                Waypoint Linea18_B: TCP in base x=-1149.609 y=625.735 z=110.055 mm, rx=1.1641 ry=-2.9058 rz=0.0105 rad; joints [-36.269, -18.655, 11.335, 7.818, -269.001, 0.894] deg; TCP offset x=0.411 y=-218.298 z=37.994 mm, rx=1.558 ry=-0.1255 rz=0.1212 rad
            Folder AB
              'desbaste_inicial'
              bajada_broca := p[0,0,-0.008,0,0,0]
              barrenos_menos1 := 19
              barreno_actual := 0
              Loop While (checkContinuously=false) expression=barreno_actual≤barrenos_menos1
                Folder Perforacion
                  MoveL speed 100 mm/s, acceleration 500 mm/s^2 (useActiveTCP=true) feature=Base
                    If barreno_actual≟6  or barreno_actual≟13
                      barreno_actual := barreno_actual+1
                    internos := interpolate_pose(Linea18_A, Linea18_B, barreno_actual/barrenos_menos1)
                    Waypoint Waypoint (Variable): variable=internos
                    'desbaste_inicial'
                    bajada_broca := p[0,0,-0.008,0,0,0]
                    bajada := p[0,0,0.008,0,0,0]
                    MoveDirectionNode (selectedDirection=ZMinus toolParams=0.1, 0.15)
                      Until DISTANCE (allowActions=false deceleration=3 distanceNodeType=STOP) Distance=0.071; motionParameters(blendRadius=0)
                    MoveDirectionNode (selectedDirection=ZMinus toolParams=0.001, 0.001)
                      Until TOOL_CONTACT_DETECTION (allowActions=false retraction=0 decelerationAcceleration=0.001 decelerationAngularAcceleration=34.906585)
                    Popup Message (haltProgram=false message=punto contacto alanzdo inputType=Text)
                    MoveDirectionNode (selectedDirection=ZPlus toolParams=0.003, 0.005)
                      Until DISTANCE (allowActions=false deceleration=3 distanceNodeType=STOP) Distance=0.002; motionParameters(blendRadius=0)
                    Wait Sleep waitTime=0.3
                    Set DigitalOutput pin=config_out[1]; digitalValue=1
                    Wait Sleep waitTime=0.3
                    SuppressedNode
                      Loop Counting (count=3) loopVariable=Loop_92
                        bajar := pose_add(get_actual_tcp_pose(), bajada_broca)
                        Waypoint Waypoint (Variable): motionParameters(jointSpeed=1.047198 jointAcceleration=1.396263 cartesianSpeed=0.001 cartesianAcceleration=0.005); variable=bajar
                        subir := pose_sub(get_actual_tcp_pose(), bajada_broca)
                        Waypoint Waypoint (Variable): motionParameters(jointSpeed=1.047198 jointAcceleration=1.396263 cartesianSpeed=0.005 cartesianAcceleration=0.01); variable=subir
                        bajada_broca := pose_sub(bajada_broca, bajada)
                    MoveDirectionNode (selectedDirection=ZPlus toolParams=0.1, 0.15)
                      Until DISTANCE (allowActions=false deceleration=3 distanceNodeType=STOP) Distance=0.08; motionParameters(blendRadius=0)
                    Set DigitalOutput pin=config_out[1]; digitalValue=0
                    barreno_actual := barreno_actual+1
                    SuppressedNode
                      Call Quitar_broca
                    SuppressedNode
                      Call Poner_broca
          Popup Message (haltProgram=false message=Linea18 con chica Terminada! inputType=Text)
      Folder Broca_1
        Folder Linea7
          Folder Marcar_puntos
            MoveL speed 100 mm/s, acceleration 500 mm/s^2 (useActiveTCP=true) feature=Base
              Waypoint Home2: TCP in base x=649.602 y=3.2 z=254.15 mm, rx=-2.4485 ry=-1.9662 rz=-0.0111 rad; joints [-199.372, -96.579, 116.673, -19.801, -286.041, 0.348] deg
              Waypoint Linea7_A: TCP in base x=737.913 y=-359.697 z=110.247 mm, rx=3.1319 ry=0.1866 rz=-0.0004 rad; joints [-210.915, -68.733, 100.688, -31.639, -226.901, 0.305] deg
              Folder bajada_comprobacion
                MoveDirectionNode (selectedDirection=ZMinus toolParams=0.1, 0.15)
                  Until DISTANCE (allowActions=false deceleration=3 distanceNodeType=STOP) Distance=0.071; motionParameters(blendRadius=0)
                MoveDirectionNode (selectedDirection=ZMinus toolParams=0.007, 0.007)
                  Until TOOL_CONTACT_DETECTION (allowActions=false retraction=0 decelerationAcceleration=0.02 decelerationAngularAcceleration=34.906585)
                MoveDirectionNode (selectedDirection=ZPlus toolParams=0.1, 0.15)
                  Until DISTANCE (allowActions=false deceleration=3 distanceNodeType=STOP) Distance=0.08; motionParameters(blendRadius=0)
              Waypoint Linea7_B: TCP in base x=783.713 y=-360.081 z=110.621 mm, rx=3.1319 ry=0.1866 rz=-0.0004 rad; joints [-209.138, -65.085, 95.206, -29.798, -225.12, 0.318] deg
              Folder bajada_comprobacion
                MoveDirectionNode (selectedDirection=ZMinus toolParams=0.1, 0.15)
                  Until DISTANCE (allowActions=false deceleration=3 distanceNodeType=STOP) Distance=0.071; motionParameters(blendRadius=0)
                MoveDirectionNode (selectedDirection=ZMinus toolParams=0.007, 0.007)
                  Until TOOL_CONTACT_DETECTION (allowActions=false retraction=0 decelerationAcceleration=0.02 decelerationAngularAcceleration=34.906585)
                MoveDirectionNode (selectedDirection=ZPlus toolParams=0.1, 0.15)
                  Until DISTANCE (allowActions=false deceleration=3 distanceNodeType=STOP) Distance=0.08; motionParameters(blendRadius=0)
          Folder AB
            'desbaste_inicial'
            bajada_broca := p[0,0,-0.008,0,0,0]
            barrenos_menos1 := 2
            barreno_actual := 1
            Loop While (checkContinuously=false) expression=barreno_actual≤barrenos_menos1
              Folder Perforacion
                MoveL speed 100 mm/s, acceleration 500 mm/s^2 (useActiveTCP=true) feature=Base
                  internos := interpolate_pose(Linea7_A, Linea7_B, barreno_actual/barrenos_menos1)
                  Waypoint Waypoint (Variable): variable=internos
                  'desbaste_inicial'
                  bajada_broca := p[0,0,-0.024,0,0,0]
                  bajada := p[0,0,0.024,0,0,0]
                  MoveDirectionNode (selectedDirection=ZMinus toolParams=0.1, 0.15)
                    Until DISTANCE (allowActions=false deceleration=3 distanceNodeType=STOP) Distance=0.071; motionParameters(blendRadius=0)
                  MoveDirectionNode (selectedDirection=ZMinus toolParams=0.007, 0.007)
                    Until TOOL_CONTACT_DETECTION (allowActions=false retraction=0 decelerationAcceleration=0.02 decelerationAngularAcceleration=34.906585)
                  Popup Message (haltProgram=false message=punto contacto alanzdo inputType=Text)
                  MoveDirectionNode (selectedDirection=ZPlus toolParams=0.015, 0.015)
                    Until DISTANCE (allowActions=false deceleration=3 distanceNodeType=STOP) Distance=0.007; motionParameters(blendRadius=0)
                  Wait Sleep waitTime=0.3
                  Set DigitalOutput pin=config_out[1]; digitalValue=1
                  Wait Sleep waitTime=0.3
                  Loop Counting (count=1) loopVariable(name=Loop_96)
                    bajar := pose_add(get_actual_tcp_pose(), bajada_broca)
                    Waypoint Waypoint (Variable): motionParameters(jointSpeed=1.047198 jointAcceleration=1.396263 cartesianSpeed=0.004 cartesianAcceleration=0.004); variable=bajar
                    subir := pose_sub(get_actual_tcp_pose(), bajada_broca)
                    MoveDirectionNode (selectedDirection=ZPlus toolParams=0.015, 0.015)
                      Until DISTANCE (allowActions=false deceleration=3 distanceNodeType=STOP) Distance=0.002; motionParameters(blendRadius=0)
                    Set DigitalOutput pin=config_out[1]; digitalValue=0
                    Waypoint Waypoint (Variable): motionParameters(jointSpeed=1.047198 jointAcceleration=1.396263 cartesianSpeed=0.015 cartesianAcceleration=0.015); variable=subir
                    bajada_broca := pose_sub(bajada_broca, bajada)
                  MoveDirectionNode (selectedDirection=ZPlus toolParams=0.1, 0.15)
                    Until DISTANCE (allowActions=false deceleration=3 distanceNodeType=STOP) Distance=0.08; motionParameters(blendRadius=0)
                  Set DigitalOutput pin=config_out[1]; digitalValue=0
                  barreno_actual := barreno_actual+1
                  Call Quitar_broca
                  Call Poner_broca
        Popup Message (haltProgram=false message=Linea7 con chica Terminada! inputType=Text)
        Folder Linea8
          Folder Marcar_puntos
            MoveL speed 100 mm/s, acceleration 500 mm/s^2 (useActiveTCP=true) feature=Base
              Waypoint Linea8_A: TCP in base x=886.283 y=-360.229 z=110.454 mm, rx=3.1315 ry=0.1865 rz=0.0006 rad; joints [-205.767, -56.675, 81.874, -24.901, -221.735, 0.344] deg
              Folder bajada_comprobacion
                MoveDirectionNode (selectedDirection=ZMinus toolParams=0.1, 0.15)
                  Until DISTANCE (allowActions=false deceleration=3 distanceNodeType=STOP) Distance=0.071; motionParameters(blendRadius=0)
                MoveDirectionNode (selectedDirection=ZMinus toolParams=0.007, 0.007)
                  Until TOOL_CONTACT_DETECTION (allowActions=false retraction=0 decelerationAcceleration=0.02 decelerationAngularAcceleration=34.906585)
                MoveDirectionNode (selectedDirection=ZPlus toolParams=0.1, 0.15)
                  Until DISTANCE (allowActions=false deceleration=3 distanceNodeType=STOP) Distance=0.08; motionParameters(blendRadius=0)
              Waypoint Linea8_B: TCP in base x=1009.987 y=-360.229 z=110.179 mm, rx=3.1315 ry=0.1865 rz=0.0006 rad; joints [-202.59, -45.403, 62.493, -16.778, -218.539, 0.367] deg
              Folder bajada_comprobacion
                MoveDirectionNode (selectedDirection=ZMinus toolParams=0.1, 0.15)
                  Until DISTANCE (allowActions=false deceleration=3 distanceNodeType=STOP) Distance=0.071; motionParameters(blendRadius=0)
                MoveDirectionNode (selectedDirection=ZMinus toolParams=0.007, 0.007)
                  Until TOOL_CONTACT_DETECTION (allowActions=false retraction=0 decelerationAcceleration=0.02 decelerationAngularAcceleration=34.906585)
                MoveDirectionNode (selectedDirection=ZPlus toolParams=0.1, 0.15)
                  Until DISTANCE (allowActions=false deceleration=3 distanceNodeType=STOP) Distance=0.08; motionParameters(blendRadius=0)
          Folder AB
            'desbaste_inicial'
            bajada_broca := p[0,0,-0.008,0,0,0]
            barrenos_menos1 := 5
            barreno_actual := 0
            Loop While (checkContinuously=false) expression=barreno_actual≤barrenos_menos1
              Folder Perforacion
                MoveL speed 100 mm/s, acceleration 500 mm/s^2 (useActiveTCP=true) feature=Base
                  internos := interpolate_pose(Linea8_A, Linea8_B, barreno_actual/barrenos_menos1)
                  Waypoint Waypoint (Variable): variable=internos
                  'desbaste_inicial'
                  bajada_broca := p[0,0,-0.024,0,0,0]
                  bajada := p[0,0,0.0024,0,0,0]
                  MoveDirectionNode (selectedDirection=ZMinus toolParams=0.1, 0.15)
                    Until DISTANCE (allowActions=false deceleration=3 distanceNodeType=STOP) Distance=0.071; motionParameters(blendRadius=0)
                  MoveDirectionNode (selectedDirection=ZMinus toolParams=0.007, 0.007)
                    Until TOOL_CONTACT_DETECTION (allowActions=false retraction=0 decelerationAcceleration=0.02 decelerationAngularAcceleration=34.906585)
                  Popup Message (haltProgram=false message=punto contacto alanzdo inputType=Text)
                  MoveDirectionNode (selectedDirection=ZPlus toolParams=0.015, 0.015)
                    Until DISTANCE (allowActions=false deceleration=3 distanceNodeType=STOP) Distance=0.007; motionParameters(blendRadius=0)
                  Wait Sleep waitTime=0.3
                  Set DigitalOutput pin=config_out[1]; digitalValue=1
                  Wait Sleep waitTime=0.3
                  Loop Counting (count=1) loopVariable(name=Loop_110)
                    bajar := pose_add(get_actual_tcp_pose(), bajada_broca)
                    Waypoint Waypoint (Variable): motionParameters(jointSpeed=1.047198 jointAcceleration=1.396263 cartesianSpeed=0.004 cartesianAcceleration=0.004); variable=bajar
                    subir := pose_sub(get_actual_tcp_pose(), bajada_broca)
                    MoveDirectionNode (selectedDirection=ZPlus toolParams=0.015, 0.015)
                      Until DISTANCE (allowActions=false deceleration=3 distanceNodeType=STOP) Distance=0.002; motionParameters(blendRadius=0)
                    Set DigitalOutput pin=config_out[1]; digitalValue=0
                    Waypoint Waypoint (Variable): motionParameters(jointSpeed=1.047198 jointAcceleration=1.396263 cartesianSpeed=0.015 cartesianAcceleration=0.015); variable=subir
                    bajada_broca := pose_sub(bajada_broca, bajada)
                  MoveDirectionNode (selectedDirection=ZPlus toolParams=0.1, 0.15)
                    Until DISTANCE (allowActions=false deceleration=3 distanceNodeType=STOP) Distance=0.08; motionParameters(blendRadius=0)
                  Set DigitalOutput pin=config_out[1]; digitalValue=0
                  barreno_actual := barreno_actual+1
                  Call Quitar_broca
                  Call Poner_broca
        Popup Message (haltProgram=false message=Linea8 con chica Terminada! inputType=Text)
        Folder Linea9
          Folder Marcar_puntos
            MoveL speed 100 mm/s, acceleration 500 mm/s^2 (useActiveTCP=true) feature=Base
              Waypoint Linea9_A: TCP in base x=1089.313 y=-360.631 z=110.237 mm, rx=3.1313 ry=0.1866 rz=0.0014 rad; joints [-200.952, -36.589, 46.349, -9.474, -216.885, 0.379] deg
              Folder bajada_comprobacion
                MoveDirectionNode (selectedDirection=ZMinus toolParams=0.1, 0.15)
                  Until DISTANCE (allowActions=false deceleration=3 distanceNodeType=STOP) Distance=0.071; motionParameters(blendRadius=0)
                MoveDirectionNode (selectedDirection=ZMinus toolParams=0.007, 0.007)
                  Until TOOL_CONTACT_DETECTION (allowActions=false retraction=0 decelerationAcceleration=0.02 decelerationAngularAcceleration=34.906585)
                MoveDirectionNode (selectedDirection=ZPlus toolParams=0.1, 0.15)
                  Until DISTANCE (allowActions=false deceleration=3 distanceNodeType=STOP) Distance=0.08; motionParameters(blendRadius=0)
              Waypoint Linea9_B: TCP in base x=1138.944 y=-360.869 z=110.826 mm, rx=3.1313 ry=0.1866 rz=0.0014 rad; joints [-200.044, -29.362, 32.524, -2.871, -215.958, 0.386] deg
              Folder bajada_comprobacion
                MoveDirectionNode (selectedDirection=ZMinus toolParams=0.1, 0.15)
                  Until DISTANCE (allowActions=false deceleration=3 distanceNodeType=STOP) Distance=0.071; motionParameters(blendRadius=0)
                MoveDirectionNode (selectedDirection=ZMinus toolParams=0.007, 0.007)
                  Until TOOL_CONTACT_DETECTION (allowActions=false retraction=0 decelerationAcceleration=0.02 decelerationAngularAcceleration=34.906585)
                MoveDirectionNode (selectedDirection=ZPlus toolParams=0.1, 0.15)
                  Until DISTANCE (allowActions=false deceleration=3 distanceNodeType=STOP) Distance=0.08; motionParameters(blendRadius=0)
          Folder AB
            'desbaste_inicial'
            bajada_broca := p[0,0,-0.008,0,0,0]
            barrenos_menos1 := 2
            barreno_actual := 0
            Loop While (checkContinuously=false) expression=barreno_actual≤barrenos_menos1
              Folder Perforacion
                MoveL speed 100 mm/s, acceleration 500 mm/s^2 (useActiveTCP=true) feature=Base
                  internos := interpolate_pose(Linea9_A, Linea9_B, barreno_actual/barrenos_menos1)
                  Waypoint Waypoint (Variable): variable=internos
                  'desbaste_inicial'
                  bajada_broca := p[0,0,-0.024,0,0,0]
                  bajada := p[0,0,0.024,0,0,0]
                  MoveDirectionNode (selectedDirection=ZMinus toolParams=0.1, 0.15)
                    Until DISTANCE (allowActions=false deceleration=3 distanceNodeType=STOP) Distance=0.071; motionParameters(blendRadius=0)
                  MoveDirectionNode (selectedDirection=ZMinus toolParams=0.007, 0.007)
                    Until TOOL_CONTACT_DETECTION (allowActions=false retraction=0 decelerationAcceleration=0.02 decelerationAngularAcceleration=34.906585)
                  Popup Message (haltProgram=false message=punto contacto alanzdo inputType=Text)
                  MoveDirectionNode (selectedDirection=ZPlus toolParams=0.015, 0.015)
                    Until DISTANCE (allowActions=false deceleration=3 distanceNodeType=STOP) Distance=0.007; motionParameters(blendRadius=0)
                  Wait Sleep waitTime=0.3
                  Set DigitalOutput pin=config_out[1]; digitalValue=1
                  Wait Sleep waitTime=0.3
                  Loop Counting (count=1) loopVariable(name=Loop_114)
                    bajar := pose_add(get_actual_tcp_pose(), bajada_broca)
                    Waypoint Waypoint (Variable): motionParameters(jointSpeed=1.047198 jointAcceleration=1.396263 cartesianSpeed=0.004 cartesianAcceleration=0.004); variable=bajar
                    subir := pose_sub(get_actual_tcp_pose(), bajada_broca)
                    MoveDirectionNode (selectedDirection=ZPlus toolParams=0.015, 0.015)
                      Until DISTANCE (allowActions=false deceleration=3 distanceNodeType=STOP) Distance=0.002; motionParameters(blendRadius=0)
                    Set DigitalOutput pin=config_out[1]; digitalValue=0
                    Waypoint Waypoint (Variable): motionParameters(jointSpeed=1.047198 jointAcceleration=1.396263 cartesianSpeed=0.015 cartesianAcceleration=0.015); variable=subir
                    bajada_broca := pose_sub(bajada_broca, bajada)
                  MoveDirectionNode (selectedDirection=ZPlus toolParams=0.1, 0.15)
                    Until DISTANCE (allowActions=false deceleration=3 distanceNodeType=STOP) Distance=0.08; motionParameters(blendRadius=0)
                  Set DigitalOutput pin=config_out[1]; digitalValue=0
                  barreno_actual := barreno_actual+1
                  Call Quitar_broca
                  Call Poner_broca
        Popup Message (haltProgram=false message=Linea9 con chica Terminada! inputType=Text)
        Folder Linea10
          Folder Marcar_puntos
            MoveL speed 100 mm/s, acceleration 500 mm/s^2 (useActiveTCP=true) feature=Base
              Waypoint Home2: TCP in base x=649.602 y=3.2 z=254.15 mm, rx=-2.4485 ry=-1.9662 rz=-0.0111 rad; joints [-199.372, -96.579, 116.673, -19.801, -286.041, 0.348] deg
              Waypoint Linea10_A: TCP in base x=620.978 y=-324.892 z=110.624 mm, rx=3.1274 ry=-0.2451 rz=-0.0041 rad; joints [-211.246, -75.766, 110.43, -34.284, -211.451, 0.322] deg; TCP offset x=0.411 y=-218.298 z=37.994 mm, rx=1.558 ry=-0.1255 rz=0.1212 rad
              Folder bajada_comprobacion
                MoveDirectionNode (selectedDirection=ZMinus toolParams=0.1, 0.15)
                  Until DISTANCE (allowActions=false deceleration=3 distanceNodeType=STOP) Distance=0.071; motionParameters(blendRadius=0)
                MoveDirectionNode (selectedDirection=ZMinus toolParams=0.007, 0.007)
                  Until TOOL_CONTACT_DETECTION (allowActions=false retraction=0 decelerationAcceleration=0.02 decelerationAngularAcceleration=34.906585)
                MoveDirectionNode (selectedDirection=ZPlus toolParams=0.1, 0.15)
                  Until DISTANCE (allowActions=false deceleration=3 distanceNodeType=STOP) Distance=0.08; motionParameters(blendRadius=0)
              Waypoint Linea10_B: TCP in base x=621.098 y=-276.98 z=110.32 mm, rx=3.1274 ry=-0.2451 rz=-0.0041 rad; joints [-207.342, -76.685, 111.673, -34.563, -207.548, 0.378] deg
              Folder bajada_comprobacion
                MoveDirectionNode (selectedDirection=ZMinus toolParams=0.1, 0.15)
                  Until DISTANCE (allowActions=false deceleration=3 distanceNodeType=STOP) Distance=0.071; motionParameters(blendRadius=0)
                MoveDirectionNode (selectedDirection=ZMinus toolParams=0.007, 0.007)
                  Until TOOL_CONTACT_DETECTION (allowActions=false retraction=0 decelerationAcceleration=0.02 decelerationAngularAcceleration=34.906585)
                MoveDirectionNode (selectedDirection=ZPlus toolParams=0.1, 0.15)
                  Until DISTANCE (allowActions=false deceleration=3 distanceNodeType=STOP) Distance=0.08; motionParameters(blendRadius=0)
          Folder AB
            'desbaste_inicial'
            bajada_broca := p[0,0,-0.008,0,0,0]
            barrenos_menos1 := 2
            barreno_actual := 0
            Loop While (checkContinuously=false) expression=barreno_actual≤barrenos_menos1
              Folder Perforacion
                MoveL speed 100 mm/s, acceleration 500 mm/s^2 (useActiveTCP=true) feature=Base
                  internos := interpolate_pose(Linea10_A, Linea10_B, barreno_actual/barrenos_menos1)
                  Waypoint Waypoint (Variable): variable=internos
                  'desbaste_inicial'
                  bajada_broca := p[0,0,-0.024,0,0,0]
                  bajada := p[0,0,0.024,0,0,0]
                  MoveDirectionNode (selectedDirection=ZMinus toolParams=0.1, 0.15)
                    Until DISTANCE (allowActions=false deceleration=3 distanceNodeType=STOP) Distance=0.071; motionParameters(blendRadius=0)
                  MoveDirectionNode (selectedDirection=ZMinus toolParams=0.007, 0.007)
                    Until TOOL_CONTACT_DETECTION (allowActions=false retraction=0 decelerationAcceleration=0.02 decelerationAngularAcceleration=34.906585)
                  Popup Message (haltProgram=false message=punto contacto alanzdo inputType=Text)
                  MoveDirectionNode (selectedDirection=ZPlus toolParams=0.015, 0.015)
                    Until DISTANCE (allowActions=false deceleration=3 distanceNodeType=STOP) Distance=0.007; motionParameters(blendRadius=0)
                  Wait Sleep waitTime=0.3
                  Set DigitalOutput pin=config_out[1]; digitalValue=1
                  Wait Sleep waitTime=0.3
                  Loop Counting (count=1) loopVariable(name=Loop_118)
                    bajar := pose_add(get_actual_tcp_pose(), bajada_broca)
                    Waypoint Waypoint (Variable): motionParameters(jointSpeed=1.047198 jointAcceleration=1.396263 cartesianSpeed=0.004 cartesianAcceleration=0.004); variable=bajar
                    subir := pose_sub(get_actual_tcp_pose(), bajada_broca)
                    MoveDirectionNode (selectedDirection=ZPlus toolParams=0.015, 0.015)
                      Until DISTANCE (allowActions=false deceleration=3 distanceNodeType=STOP) Distance=0.002; motionParameters(blendRadius=0)
                    Set DigitalOutput pin=config_out[1]; digitalValue=0
                    Waypoint Waypoint (Variable): motionParameters(jointSpeed=1.047198 jointAcceleration=1.396263 cartesianSpeed=0.015 cartesianAcceleration=0.015); variable=subir
                    bajada_broca := pose_sub(bajada_broca, bajada)
                  MoveDirectionNode (selectedDirection=ZPlus toolParams=0.1, 0.15)
                    Until DISTANCE (allowActions=false deceleration=3 distanceNodeType=STOP) Distance=0.08; motionParameters(blendRadius=0)
                  Set DigitalOutput pin=config_out[1]; digitalValue=0
                  barreno_actual := barreno_actual+1
                  SuppressedNode
                    Call Quitar_broca
                  SuppressedNode
                    Call Poner_broca
        Popup Message (haltProgram=false message=Linea10 con chica Terminada! inputType=Text)
        Folder Linea11
          Folder Marcar_puntos
            MoveL speed 100 mm/s, acceleration 500 mm/s^2 (useActiveTCP=true) feature=Base
              Waypoint Linea11_A: TCP in base x=623.455 y=-144.673 z=110.191 mm, rx=-2.632 ry=-1.7105 rz=-0.0086 rad; joints [-213.683, -89.957, 126.956, -36.551, -288.892, 0.32] deg
              Folder bajada_comprobacion
                MoveDirectionNode (selectedDirection=ZMinus toolParams=0.1, 0.15)
                  Until DISTANCE (allowActions=false deceleration=3 distanceNodeType=STOP) Distance=0.071; motionParameters(blendRadius=0)
                MoveDirectionNode (selectedDirection=ZMinus toolParams=0.007, 0.007)
                  Until TOOL_CONTACT_DETECTION (allowActions=false retraction=0 decelerationAcceleration=0.02 decelerationAngularAcceleration=34.906585)
                MoveDirectionNode (selectedDirection=ZPlus toolParams=0.1, 0.15)
                  Until DISTANCE (allowActions=false deceleration=3 distanceNodeType=STOP) Distance=0.08; motionParameters(blendRadius=0)
              Waypoint Linea11_B: TCP in base x=624.12 y=-90.095 z=110.354 mm, rx=-2.632 ry=-1.7105 rz=-0.0086 rad; joints [-207.683, -90.822, 127.793, -36.543, -282.892, 0.367] deg
              Folder bajada_comprobacion
                MoveDirectionNode (selectedDirection=ZMinus toolParams=0.1, 0.15)
                  Until DISTANCE (allowActions=false deceleration=3 distanceNodeType=STOP) Distance=0.071; motionParameters(blendRadius=0)
                MoveDirectionNode (selectedDirection=ZMinus toolParams=0.007, 0.007)
                  Until TOOL_CONTACT_DETECTION (allowActions=false retraction=0 decelerationAcceleration=0.02 decelerationAngularAcceleration=34.906585)
                MoveDirectionNode (selectedDirection=ZPlus toolParams=0.1, 0.15)
                  Until DISTANCE (allowActions=false deceleration=3 distanceNodeType=STOP) Distance=0.08; motionParameters(blendRadius=0)
          Folder AB
            'desbaste_inicial'
            bajada_broca := p[0,0,-0.008,0,0,0]
            barrenos_menos1 := 2
            barreno_actual := 0
            Loop While (checkContinuously=false) expression=barreno_actual≤barrenos_menos1
              Folder Perforacion
                MoveL speed 100 mm/s, acceleration 500 mm/s^2 (useActiveTCP=true) feature=Base
                  SuppressedNode
                    If barreno_actual≟5
                      barreno_actual := barreno_actual+1
                  internos := interpolate_pose(Linea11_A, Linea11_B, barreno_actual/barrenos_menos1)
                  Waypoint Waypoint (Variable): variable=internos
                  'desbaste_inicial'
                  bajada_broca := p[0,0,-0.024,0,0,0]
                  bajada := p[0,0,0.024,0,0,0]
                  MoveDirectionNode (selectedDirection=ZMinus toolParams=0.1, 0.15)
                    Until DISTANCE (allowActions=false deceleration=3 distanceNodeType=STOP) Distance=0.071; motionParameters(blendRadius=0)
                  MoveDirectionNode (selectedDirection=ZMinus toolParams=0.007, 0.007)
                    Until TOOL_CONTACT_DETECTION (allowActions=false retraction=0 decelerationAcceleration=0.02 decelerationAngularAcceleration=34.906585)
                  Popup Message (haltProgram=false message=punto contacto alanzdo inputType=Text)
                  MoveDirectionNode (selectedDirection=ZPlus toolParams=0.015, 0.015)
                    Until DISTANCE (allowActions=false deceleration=3 distanceNodeType=STOP) Distance=0.007; motionParameters(blendRadius=0)
                  Wait Sleep waitTime=0.3
                  Set DigitalOutput pin=config_out[1]; digitalValue=1
                  Wait Sleep waitTime=0.3
                  Loop Counting (count=1) loopVariable(name=Loop_122)
                    bajar := pose_add(get_actual_tcp_pose(), bajada_broca)
                    Waypoint Waypoint (Variable): motionParameters(jointSpeed=1.047198 jointAcceleration=1.396263 cartesianSpeed=0.004 cartesianAcceleration=0.004); variable=bajar
                    subir := pose_sub(get_actual_tcp_pose(), bajada_broca)
                    MoveDirectionNode (selectedDirection=ZPlus toolParams=0.015, 0.015)
                      Until DISTANCE (allowActions=false deceleration=3 distanceNodeType=STOP) Distance=0.002; motionParameters(blendRadius=0)
                    Set DigitalOutput pin=config_out[1]; digitalValue=0
                    Waypoint Waypoint (Variable): motionParameters(jointSpeed=1.047198 jointAcceleration=1.396263 cartesianSpeed=0.015 cartesianAcceleration=0.015); variable=subir
                    bajada_broca := pose_sub(bajada_broca, bajada)
                  MoveDirectionNode (selectedDirection=ZPlus toolParams=0.1, 0.15)
                    Until DISTANCE (allowActions=false deceleration=3 distanceNodeType=STOP) Distance=0.08; motionParameters(blendRadius=0)
                  Set DigitalOutput pin=config_out[1]; digitalValue=0
                  barreno_actual := barreno_actual+1
                  SuppressedNode
                    Call Quitar_broca
                  SuppressedNode
                    Call Poner_broca
        Popup Message (haltProgram=false message=Linea11 con chica Terminada! inputType=Text)
        Folder Linea12
          Folder Marcar_puntos
            MoveL speed 100 mm/s, acceleration 500 mm/s^2 (useActiveTCP=true) feature=Base
              Waypoint Linea12_A: TCP in base x=624.141 y=-66.274 z=110.335 mm, rx=-2.6321 ry=-1.7106 rz=-0.0087 rad; joints [-204.939, -91.033, 128.004, -36.559, -280.152, 0.387] deg
              Folder bajada_comprobacion
                MoveDirectionNode (selectedDirection=ZMinus toolParams=0.1, 0.15)
                  Until DISTANCE (allowActions=false deceleration=3 distanceNodeType=STOP) Distance=0.071; motionParameters(blendRadius=0)
                MoveDirectionNode (selectedDirection=ZMinus toolParams=0.007, 0.007)
                  Until TOOL_CONTACT_DETECTION (allowActions=false retraction=0 decelerationAcceleration=0.02 decelerationAngularAcceleration=34.906585)
                MoveDirectionNode (selectedDirection=ZPlus toolParams=0.1, 0.15)
                  Until DISTANCE (allowActions=false deceleration=3 distanceNodeType=STOP) Distance=0.08; motionParameters(blendRadius=0)
              Waypoint Linea12_B: TCP in base x=625.005 y=106.664 z=110.181 mm, rx=-2.6321 ry=-1.7106 rz=-0.0087 rad; joints [-183.741, -88.918, 125.907, -36.601, -258.955, 0.536] deg
              Folder bajada_comprobacion
                MoveDirectionNode (selectedDirection=ZMinus toolParams=0.1, 0.15)
                  Until DISTANCE (allowActions=false deceleration=3 distanceNodeType=STOP) Distance=0.071; motionParameters(blendRadius=0)
                MoveDirectionNode (selectedDirection=ZMinus toolParams=0.007, 0.007)
                  Until TOOL_CONTACT_DETECTION (allowActions=false retraction=0 decelerationAcceleration=0.02 decelerationAngularAcceleration=34.906585)
                MoveDirectionNode (selectedDirection=ZPlus toolParams=0.1, 0.15)
                  Until DISTANCE (allowActions=false deceleration=3 distanceNodeType=STOP) Distance=0.08; motionParameters(blendRadius=0)
          Folder AB
            'desbaste_inicial'
            bajada_broca := p[0,0,-0.008,0,0,0]
            barrenos_menos1 := 7
            barreno_actual := 0
            Loop While (checkContinuously=false) expression=barreno_actual≤barrenos_menos1
              Folder Perforacion
                MoveL speed 100 mm/s, acceleration 500 mm/s^2 (useActiveTCP=true) feature=Base
                  If barreno_actual≟2
                    barreno_actual := barreno_actual+1
                  internos := interpolate_pose(Linea12_A, Linea12_B, barreno_actual/barrenos_menos1)
                  Waypoint Waypoint (Variable): variable=internos
                  'desbaste_inicial'
                  bajada_broca := p[0,0,-0.024,0,0,0]
                  bajada := p[0,0,0.024,0,0,0]
                  MoveDirectionNode (selectedDirection=ZMinus toolParams=0.1, 0.15)
                    Until DISTANCE (allowActions=false deceleration=3 distanceNodeType=STOP) Distance=0.071; motionParameters(blendRadius=0)
                  MoveDirectionNode (selectedDirection=ZMinus toolParams=0.007, 0.007)
                    Until TOOL_CONTACT_DETECTION (allowActions=false retraction=0 decelerationAcceleration=0.02 decelerationAngularAcceleration=34.906585)
                  Popup Message (haltProgram=false message=punto contacto alanzdo inputType=Text)
                  MoveDirectionNode (selectedDirection=ZPlus toolParams=0.015, 0.015)
                    Until DISTANCE (allowActions=false deceleration=3 distanceNodeType=STOP) Distance=0.002; motionParameters(blendRadius=0)
                  Wait Sleep waitTime=0.3
                  Set DigitalOutput pin=config_out[1]; digitalValue=1
                  Wait Sleep waitTime=0.3
                  Loop Counting (count=1) loopVariable(name=Loop_126)
                    bajar := pose_add(get_actual_tcp_pose(), bajada_broca)
                    Waypoint Waypoint (Variable): motionParameters(jointSpeed=1.047198 jointAcceleration=1.396263 cartesianSpeed=0.004 cartesianAcceleration=0.004); variable=bajar
                    subir := pose_sub(get_actual_tcp_pose(), bajada_broca)
                    MoveDirectionNode (selectedDirection=ZPlus toolParams=0.015, 0.015)
                      Until DISTANCE (allowActions=false deceleration=3 distanceNodeType=STOP) Distance=0.002; motionParameters(blendRadius=0)
                    Set DigitalOutput pin=config_out[1]; digitalValue=0
                    Waypoint Waypoint (Variable): motionParameters(jointSpeed=1.047198 jointAcceleration=1.396263 cartesianSpeed=0.015 cartesianAcceleration=0.015); variable=subir
                    bajada_broca := pose_sub(bajada_broca, bajada)
                  MoveDirectionNode (selectedDirection=ZPlus toolParams=0.1, 0.15)
                    Until DISTANCE (allowActions=false deceleration=3 distanceNodeType=STOP) Distance=0.08; motionParameters(blendRadius=0)
                  Set DigitalOutput pin=config_out[1]; digitalValue=0
                  barreno_actual := barreno_actual+1
                  SuppressedNode
                    Call Quitar_broca
                  SuppressedNode
                    Call Poner_broca
        Popup Message (haltProgram=false message=Linea12 con chica Terminada! inputType=Text)
        Folder Linea13
          Folder Marcar_puntos
            MoveL speed 100 mm/s, acceleration 500 mm/s^2 (useActiveTCP=true) feature=Base
              Waypoint Linea13_A: TCP in base x=625.493 y=262.479 z=110.355 mm, rx=-2.6325 ry=-1.7109 rz=-0.0101 rad; joints [-165.949, -82.781, 119.173, -36.043, -241.164, 0.656] deg
              Folder bajada_comprobacion
                MoveDirectionNode (selectedDirection=ZMinus toolParams=0.1, 0.15)
                  Until DISTANCE (allowActions=false deceleration=3 distanceNodeType=STOP) Distance=0.071; motionParameters(blendRadius=0)
                MoveDirectionNode (selectedDirection=ZMinus toolParams=0.007, 0.007)
                  Until TOOL_CONTACT_DETECTION (allowActions=false retraction=0 decelerationAcceleration=0.02 decelerationAngularAcceleration=34.906585)
                MoveDirectionNode (selectedDirection=ZPlus toolParams=0.1, 0.15)
                  Until DISTANCE (allowActions=false deceleration=3 distanceNodeType=STOP) Distance=0.08; motionParameters(blendRadius=0)
              Waypoint Linea13_B: TCP in base x=625.493 y=318.857 z=110.132 mm, rx=-2.6325 ry=-1.7109 rz=-0.0101 rad; joints [-160.355, -79.919, 115.767, -35.483, -235.569, 0.699] deg
              Folder bajada_comprobacion
                MoveDirectionNode (selectedDirection=ZMinus toolParams=0.1, 0.15)
                  Until DISTANCE (allowActions=false deceleration=3 distanceNodeType=STOP) Distance=0.071; motionParameters(blendRadius=0)
                MoveDirectionNode (selectedDirection=ZMinus toolParams=0.007, 0.007)
                  Until TOOL_CONTACT_DETECTION (allowActions=false retraction=0 decelerationAcceleration=0.02 decelerationAngularAcceleration=34.906585)
                MoveDirectionNode (selectedDirection=ZPlus toolParams=0.1, 0.15)
                  Until DISTANCE (allowActions=false deceleration=3 distanceNodeType=STOP) Distance=0.08; motionParameters(blendRadius=0)
          Folder AB
            'desbaste_inicial'
            bajada_broca := p[0,0,-0.008,0,0,0]
            barrenos_menos1 := 2
            barreno_actual := 0
            Loop While (checkContinuously=false) expression=barreno_actual≤barrenos_menos1
              Folder Perforacion
                MoveL speed 100 mm/s, acceleration 500 mm/s^2 (useActiveTCP=true) feature=Base
                  SuppressedNode
                    If barreno_actual≟2
                      barreno_actual := barreno_actual+1
                  internos := interpolate_pose(Linea13_A, Linea13_B, barreno_actual/barrenos_menos1)
                  Waypoint Waypoint (Variable): variable=internos
                  'desbaste_inicial'
                  bajada_broca := p[0,0,-0.024,0,0,0]
                  bajada := p[0,0,0.024,0,0,0]
                  MoveDirectionNode (selectedDirection=ZMinus toolParams=0.1, 0.15)
                    Until DISTANCE (allowActions=false deceleration=3 distanceNodeType=STOP) Distance=0.071; motionParameters(blendRadius=0)
                  MoveDirectionNode (selectedDirection=ZMinus toolParams=0.007, 0.007)
                    Until TOOL_CONTACT_DETECTION (allowActions=false retraction=0 decelerationAcceleration=0.02 decelerationAngularAcceleration=34.906585)
                  Popup Message (haltProgram=false message=punto contacto alanzdo inputType=Text)
                  MoveDirectionNode (selectedDirection=ZPlus toolParams=0.015, 0.015)
                    Until DISTANCE (allowActions=false deceleration=3 distanceNodeType=STOP) Distance=0.002; motionParameters(blendRadius=0)
                  Wait Sleep waitTime=0.3
                  Set DigitalOutput pin=config_out[1]; digitalValue=1
                  Wait Sleep waitTime=0.3
                  Loop Counting (count=1) loopVariable(name=Loop_129)
                    bajar := pose_add(get_actual_tcp_pose(), bajada_broca)
                    Waypoint Waypoint (Variable): motionParameters(jointSpeed=1.047198 jointAcceleration=1.396263 cartesianSpeed=0.004 cartesianAcceleration=0.004); variable=bajar
                    subir := pose_sub(get_actual_tcp_pose(), bajada_broca)
                    MoveDirectionNode (selectedDirection=ZPlus toolParams=0.015, 0.015)
                      Until DISTANCE (allowActions=false deceleration=3 distanceNodeType=STOP) Distance=0.002; motionParameters(blendRadius=0)
                    Set DigitalOutput pin=config_out[1]; digitalValue=0
                    Waypoint Waypoint (Variable): motionParameters(jointSpeed=1.047198 jointAcceleration=1.396263 cartesianSpeed=0.015 cartesianAcceleration=0.015); variable=subir
                    bajada_broca := pose_sub(bajada_broca, bajada)
                  MoveDirectionNode (selectedDirection=ZPlus toolParams=0.1, 0.15)
                    Until DISTANCE (allowActions=false deceleration=3 distanceNodeType=STOP) Distance=0.08; motionParameters(blendRadius=0)
                  Set DigitalOutput pin=config_out[1]; digitalValue=0
                  barreno_actual := barreno_actual+1
                  SuppressedNode
                    Call Quitar_broca
                  SuppressedNode
                    Call Poner_broca
        Popup Message (haltProgram=false message=Linea13 con chica Terminada! inputType=Text)
        Folder Linea14
          Folder Marcar_puntos
            MoveL speed 100 mm/s, acceleration 500 mm/s^2 (useActiveTCP=true) feature=Base
              Waypoint Linea14_A: TCP in base x=625.749 y=343.505 z=110.091 mm, rx=-2.6326 ry=-1.7111 rz=-0.011 rad; joints [-158.078, -78.594, 114.13, -35.197, -233.295, 0.717] deg
              barrenos_hechos := 0
              Folder bajada_comprobacion
                MoveDirectionNode (selectedDirection=ZMinus toolParams=0.1, 0.15)
                  Until DISTANCE (allowActions=false deceleration=3 distanceNodeType=STOP) Distance=0.071; motionParameters(blendRadius=0)
                MoveDirectionNode (selectedDirection=ZMinus toolParams=0.007, 0.007)
                  Until TOOL_CONTACT_DETECTION (allowActions=false retraction=0 decelerationAcceleration=0.02 decelerationAngularAcceleration=34.906585)
                MoveDirectionNode (selectedDirection=ZPlus toolParams=0.1, 0.15)
                  Until DISTANCE (allowActions=false deceleration=3 distanceNodeType=STOP) Distance=0.08; motionParameters(blendRadius=0)
              Waypoint Linea14_B: TCP in base x=626.023 y=485.153 z=110.594 mm, rx=-2.6326 ry=-1.7111 rz=-0.011 rad; joints [-146.753, -70.37, 102.998, -32.234, -221.967, 0.818] deg
              Folder bajada_comprobacion
                MoveDirectionNode (selectedDirection=ZMinus toolParams=0.1, 0.15)
                  Until DISTANCE (allowActions=false deceleration=3 distanceNodeType=STOP) Distance=0.071; motionParameters(blendRadius=0)
                MoveDirectionNode (selectedDirection=ZMinus toolParams=0.007, 0.007)
                  Until TOOL_CONTACT_DETECTION (allowActions=false retraction=0 decelerationAcceleration=0.02 decelerationAngularAcceleration=34.906585)
                MoveDirectionNode (selectedDirection=ZPlus toolParams=0.1, 0.15)
                  Until DISTANCE (allowActions=false deceleration=3 distanceNodeType=STOP) Distance=0.08; motionParameters(blendRadius=0)
          Folder AB
            'desbaste_inicial'
            bajada_broca := p[0,0,-0.008,0,0,0]
            barrenos_menos1 := 5
            barreno_actual := 0
            Loop While (checkContinuously=false) expression=barreno_actual≤barrenos_menos1
              Folder Perforacion
                MoveL speed 100 mm/s, acceleration 500 mm/s^2 (useActiveTCP=true) feature=Base
                  If barreno_actual≟3
                    barreno_actual := barreno_actual+1
                  internos := interpolate_pose(Linea14_A, Linea14_B, barreno_actual/barrenos_menos1)
                  Waypoint Waypoint (Variable): variable=internos
                  'desbaste_inicial'
                  bajada_broca := p[0,0,-0.024,0,0,0]
                  bajada := p[0,0,0.024,0,0,0]
                  MoveDirectionNode (selectedDirection=ZMinus toolParams=0.1, 0.15)
                    Until DISTANCE (allowActions=false deceleration=3 distanceNodeType=STOP) Distance=0.071; motionParameters(blendRadius=0)
                  MoveDirectionNode (selectedDirection=ZMinus toolParams=0.007, 0.007)
                    Until TOOL_CONTACT_DETECTION (allowActions=false retraction=0 decelerationAcceleration=0.02 decelerationAngularAcceleration=34.906585)
                  Popup Message (haltProgram=false message=punto contacto alanzdo inputType=Text)
                  MoveDirectionNode (selectedDirection=ZPlus toolParams=0.015, 0.015)
                    Until DISTANCE (allowActions=false deceleration=3 distanceNodeType=STOP) Distance=0.002; motionParameters(blendRadius=0)
                  Wait Sleep waitTime=0.3
                  Set DigitalOutput pin=config_out[1]; digitalValue=1
                  Wait Sleep waitTime=0.3
                  Loop Counting (count=1) loopVariable(name=Loop_131)
                    bajar := pose_add(get_actual_tcp_pose(), bajada_broca)
                    Waypoint Waypoint (Variable): motionParameters(jointSpeed=1.047198 jointAcceleration=1.396263 cartesianSpeed=0.004 cartesianAcceleration=0.004); variable=bajar
                    subir := pose_sub(get_actual_tcp_pose(), bajada_broca)
                    MoveDirectionNode (selectedDirection=ZPlus toolParams=0.015, 0.015)
                      Until DISTANCE (allowActions=false deceleration=3 distanceNodeType=STOP) Distance=0.002; motionParameters(blendRadius=0)
                    Set DigitalOutput pin=config_out[1]; digitalValue=0
                    Waypoint Waypoint (Variable): motionParameters(jointSpeed=1.047198 jointAcceleration=1.396263 cartesianSpeed=0.015 cartesianAcceleration=0.015); variable=subir
                    bajada_broca := pose_sub(bajada_broca, bajada)
                  MoveDirectionNode (selectedDirection=ZPlus toolParams=0.1, 0.15)
                    Until DISTANCE (allowActions=false deceleration=3 distanceNodeType=STOP) Distance=0.08; motionParameters(blendRadius=0)
                  Set DigitalOutput pin=config_out[1]; digitalValue=0
                  barreno_actual := barreno_actual+1
                  SuppressedNode
                    Call Quitar_broca
                  SuppressedNode
                    Call Poner_broca
        Popup Message (haltProgram=false message=Linea14 con chica Terminada! inputType=Text)
        Folder Linea15
          Folder Marcar_puntos
            MoveL speed 100 mm/s, acceleration 500 mm/s^2 (useActiveTCP=true) feature=Base
              Waypoint Linea15_A: TCP in base x=626.307 y=508.675 z=110.445 mm, rx=-2.6326 ry=-1.7111 rz=-0.011 rad; joints [-145.159, -68.884, 100.875, -31.585, -220.372, 0.835] deg
              barrenos_hechos := 0
              Folder bajada_comprobacion
                MoveDirectionNode (selectedDirection=ZMinus toolParams=0.1, 0.15)
                  Until DISTANCE (allowActions=false deceleration=3 distanceNodeType=STOP) Distance=0.071; motionParameters(blendRadius=0)
                MoveDirectionNode (selectedDirection=ZMinus toolParams=0.007, 0.007)
                  Until TOOL_CONTACT_DETECTION (allowActions=false retraction=0 decelerationAcceleration=0.02 decelerationAngularAcceleration=34.906585)
                MoveDirectionNode (selectedDirection=ZPlus toolParams=0.1, 0.15)
                  Until DISTANCE (allowActions=false deceleration=3 distanceNodeType=STOP) Distance=0.08; motionParameters(blendRadius=0)
              Waypoint Linea15_B: TCP in base x=626.328 y=587.416 z=110.05 mm, rx=-2.6327 ry=-1.711 rz=-0.011 rad; joints [-140.277, -63.781, 93.264, -29.039, -215.483, 0.889] deg
              Folder bajada_comprobacion
                MoveDirectionNode (selectedDirection=ZMinus toolParams=0.1, 0.15)
                  Until DISTANCE (allowActions=false deceleration=3 distanceNodeType=STOP) Distance=0.071; motionParameters(blendRadius=0)
                MoveDirectionNode (selectedDirection=ZMinus toolParams=0.007, 0.007)
                  Until TOOL_CONTACT_DETECTION (allowActions=false retraction=0 decelerationAcceleration=0.02 decelerationAngularAcceleration=34.906585)
                MoveDirectionNode (selectedDirection=ZPlus toolParams=0.1, 0.15)
                  Until DISTANCE (allowActions=false deceleration=3 distanceNodeType=STOP) Distance=0.08; motionParameters(blendRadius=0)
          Folder AB
            'desbaste_inicial'
            bajada_broca := p[0,0,-0.008,0,0,0]
            barrenos_menos1 := 3
            barreno_actual := 0
            Loop While (checkContinuously=false) expression=barreno_actual≤barrenos_menos1
              Folder Perforacion
                MoveL speed 100 mm/s, acceleration 500 mm/s^2 (useActiveTCP=true) feature=Base
                  SuppressedNode
                    If barreno_actual≟3
                      barreno_actual := barreno_actual+1
                  internos := interpolate_pose(Linea15_A, Linea15_B, barreno_actual/barrenos_menos1)
                  Waypoint Waypoint (Variable): variable=internos
                  'desbaste_inicial'
                  bajada_broca := p[0,0,-0.024,0,0,0]
                  bajada := p[0,0,0.024,0,0,0]
                  MoveDirectionNode (selectedDirection=ZMinus toolParams=0.1, 0.15)
                    Until DISTANCE (allowActions=false deceleration=3 distanceNodeType=STOP) Distance=0.071; motionParameters(blendRadius=0)
                  MoveDirectionNode (selectedDirection=ZMinus toolParams=0.007, 0.007)
                    Until TOOL_CONTACT_DETECTION (allowActions=false retraction=0 decelerationAcceleration=0.02 decelerationAngularAcceleration=34.906585)
                  Popup Message (haltProgram=false message=punto contacto alanzdo inputType=Text)
                  MoveDirectionNode (selectedDirection=ZPlus toolParams=0.015, 0.015)
                    Until DISTANCE (allowActions=false deceleration=3 distanceNodeType=STOP) Distance=0.002; motionParameters(blendRadius=0)
                  Wait Sleep waitTime=0.3
                  Set DigitalOutput pin=config_out[1]; digitalValue=1
                  Wait Sleep waitTime=0.3
                  Loop Counting (count=1) loopVariable(name=Loop_133)
                    bajar := pose_add(get_actual_tcp_pose(), bajada_broca)
                    Waypoint Waypoint (Variable): motionParameters(jointSpeed=1.047198 jointAcceleration=1.396263 cartesianSpeed=0.004 cartesianAcceleration=0.004); variable=bajar
                    subir := pose_sub(get_actual_tcp_pose(), bajada_broca)
                    MoveDirectionNode (selectedDirection=ZPlus toolParams=0.015, 0.015)
                      Until DISTANCE (allowActions=false deceleration=3 distanceNodeType=STOP) Distance=0.002; motionParameters(blendRadius=0)
                    Set DigitalOutput pin=config_out[1]; digitalValue=0
                    Waypoint Waypoint (Variable): motionParameters(jointSpeed=1.047198 jointAcceleration=1.396263 cartesianSpeed=0.015 cartesianAcceleration=0.015); variable=subir
                    bajada_broca := pose_sub(bajada_broca, bajada)
                  MoveDirectionNode (selectedDirection=ZPlus toolParams=0.1, 0.15)
                    Until DISTANCE (allowActions=false deceleration=3 distanceNodeType=STOP) Distance=0.08; motionParameters(blendRadius=0)
                  Set DigitalOutput pin=config_out[1]; digitalValue=0
                  barreno_actual := barreno_actual+1
                  SuppressedNode
                    Call Quitar_broca
                  SuppressedNode
                    Call Poner_broca
        Popup Message (haltProgram=false message=Linea15 con chica Terminada! inputType=Text)
        Folder Linea16
          Folder Marcar_puntos
            MoveL speed 100 mm/s, acceleration 500 mm/s^2 (useActiveTCP=true) feature=Base
              Waypoint Linea16_A referenceName=Linea16_A: TCP in base x=464.714 y=611.413 z=110.697 mm, rx=-1.5443 ry=-2.7321 rz=-0.0069 rad; joints [-140.663, -77.848, 113.101, -34.922, -270.882, 0.394] deg; TCP offset x=0.411 y=-218.298 z=37.994 mm, rx=1.558 ry=-0.1255 rz=0.1212 rad
              Folder bajada_comprobacion
                MoveDirectionNode (selectedDirection=ZMinus toolParams=0.1, 0.15)
                  Until DISTANCE (allowActions=false deceleration=3 distanceNodeType=STOP) Distance=0.071; motionParameters(blendRadius=0)
                MoveDirectionNode (selectedDirection=ZMinus toolParams=0.007, 0.007)
                  Until TOOL_CONTACT_DETECTION (allowActions=false retraction=0 decelerationAcceleration=0.02 decelerationAngularAcceleration=34.906585)
                MoveDirectionNode (selectedDirection=ZPlus toolParams=0.1, 0.15)
                  Until DISTANCE (allowActions=false deceleration=3 distanceNodeType=STOP) Distance=0.08; motionParameters(blendRadius=0)
              Waypoint Linea16_B: TCP in base x=487.741 y=611.018 z=110.415 mm, rx=-1.5443 ry=-2.7321 rz=-0.0069 rad; joints [-142.061, -76.715, 111.675, -34.628, -272.279, 0.386] deg
              Folder bajada_comprobacion
                MoveDirectionNode (selectedDirection=ZMinus toolParams=0.1, 0.15)
                  Until DISTANCE (allowActions=false deceleration=3 distanceNodeType=STOP) Distance=0.071; motionParameters(blendRadius=0)
                MoveDirectionNode (selectedDirection=ZMinus toolParams=0.007, 0.007)
                  Until TOOL_CONTACT_DETECTION (allowActions=false retraction=0 decelerationAcceleration=0.02 decelerationAngularAcceleration=34.906585)
                MoveDirectionNode (selectedDirection=ZPlus toolParams=0.1, 0.15)
                  Until DISTANCE (allowActions=false deceleration=3 distanceNodeType=STOP) Distance=0.08; motionParameters(blendRadius=0)
          Folder AB
            'desbaste_inicial'
            bajada_broca := p[0,0,-0.008,0,0,0]
            barrenos_menos1 := 1
            barreno_actual := 0
            Loop While (checkContinuously=false) expression=barreno_actual≤barrenos_menos1
              Folder Perforacion
                MoveL speed 100 mm/s, acceleration 500 mm/s^2 (useActiveTCP=true) feature=Base
                  SuppressedNode
                    If barreno_actual≟3
                      barreno_actual := barreno_actual+1
                  internos := interpolate_pose(Linea16_A, Linea16_B, barreno_actual/barrenos_menos1)
                  Waypoint Waypoint (Variable): variable=internos
                  'desbaste_inicial'
                  bajada_broca := p[0,0,-0.024,0,0,0]
                  bajada := p[0,0,0.024,0,0,0]
                  MoveDirectionNode (selectedDirection=ZMinus toolParams=0.1, 0.15)
                    Until DISTANCE (allowActions=false deceleration=3 distanceNodeType=STOP) Distance=0.071; motionParameters(blendRadius=0)
                  MoveDirectionNode (selectedDirection=ZMinus toolParams=0.007, 0.007)
                    Until TOOL_CONTACT_DETECTION (allowActions=false retraction=0 decelerationAcceleration=0.02 decelerationAngularAcceleration=34.906585)
                  Popup Message (haltProgram=false message=punto contacto alanzdo inputType=Text)
                  MoveDirectionNode (selectedDirection=ZPlus toolParams=0.015, 0.015)
                    Until DISTANCE (allowActions=false deceleration=3 distanceNodeType=STOP) Distance=0.007; motionParameters(blendRadius=0)
                  Wait Sleep waitTime=0.3
                  Set DigitalOutput pin=config_out[1]; digitalValue=1
                  Wait Sleep waitTime=0.3
                  Loop Counting (count=1) loopVariable(name=Loop_135)
                    bajar := pose_add(get_actual_tcp_pose(), bajada_broca)
                    Waypoint Waypoint (Variable): motionParameters(jointSpeed=1.047198 jointAcceleration=1.396263 cartesianSpeed=0.004 cartesianAcceleration=0.004); variable=bajar
                    subir := pose_sub(get_actual_tcp_pose(), bajada_broca)
                    MoveDirectionNode (selectedDirection=ZPlus toolParams=0.015, 0.015)
                      Until DISTANCE (allowActions=false deceleration=3 distanceNodeType=STOP) Distance=0.002; motionParameters(blendRadius=0)
                    Set DigitalOutput pin=config_out[1]; digitalValue=0
                    Waypoint Waypoint (Variable): motionParameters(jointSpeed=1.047198 jointAcceleration=1.396263 cartesianSpeed=0.015 cartesianAcceleration=0.015); variable=subir
                    bajada_broca := pose_sub(bajada_broca, bajada)
                  MoveDirectionNode (selectedDirection=ZPlus toolParams=0.1, 0.15)
                    Until DISTANCE (allowActions=false deceleration=3 distanceNodeType=STOP) Distance=0.08; motionParameters(blendRadius=0)
                  Set DigitalOutput pin=config_out[1]; digitalValue=0
                  barreno_actual := barreno_actual+1
                  SuppressedNode
                    Call Quitar_broca
                  SuppressedNode
                    Call Poner_broca
        Popup Message (haltProgram=false message=Linea16 con chica Terminada! inputType=Text)
        Folder Linea17
          Folder Marcar_puntos
            MoveL speed 100 mm/s, acceleration 500 mm/s^2 (useActiveTCP=true) feature=Base
              Waypoint Linea17_A: TCP in base x=517.384 y=611.103 z=110.729 mm, rx=-1.5448 ry=-2.7327 rz=-0.0099 rad; joints [-143.713, -75.238, 109.731, -34.279, -273.925, 0.383] deg
              Folder bajada_comprobacion
                MoveDirectionNode (selectedDirection=ZMinus toolParams=0.1, 0.15)
                  Until DISTANCE (allowActions=false deceleration=3 distanceNodeType=STOP) Distance=0.071; motionParameters(blendRadius=0)
                MoveDirectionNode (selectedDirection=ZMinus toolParams=0.007, 0.007)
                  Until TOOL_CONTACT_DETECTION (allowActions=false retraction=0 decelerationAcceleration=0.02 decelerationAngularAcceleration=34.906585)
                MoveDirectionNode (selectedDirection=ZPlus toolParams=0.1, 0.15)
                  Until DISTANCE (allowActions=false deceleration=3 distanceNodeType=STOP) Distance=0.08; motionParameters(blendRadius=0)
              Waypoint Linea17_B: TCP in base x=569.253 y=610.697 z=110.46 mm, rx=-1.5448 ry=-2.7327 rz=-0.0099 rad; joints [-146.385, -72.438, 105.956, -33.3, -276.596, 0.373] deg
              Folder bajada_comprobacion
                MoveDirectionNode (selectedDirection=ZMinus toolParams=0.1, 0.15)
                  Until DISTANCE (allowActions=false deceleration=3 distanceNodeType=STOP) Distance=0.071; motionParameters(blendRadius=0)
                MoveDirectionNode (selectedDirection=ZMinus toolParams=0.007, 0.007)
                  Until TOOL_CONTACT_DETECTION (allowActions=false retraction=0 decelerationAcceleration=0.02 decelerationAngularAcceleration=34.906585)
                MoveDirectionNode (selectedDirection=ZPlus toolParams=0.1, 0.15)
                  Until DISTANCE (allowActions=false deceleration=3 distanceNodeType=STOP) Distance=0.08; motionParameters(blendRadius=0)
          Folder AB
            'desbaste_inicial'
            bajada_broca := p[0,0,-0.008,0,0,0]
            barrenos_menos1 := 2
            barreno_actual := 0
            Loop While (checkContinuously=false) expression=barreno_actual≤barrenos_menos1
              Folder Perforacion
                MoveL speed 100 mm/s, acceleration 500 mm/s^2 (useActiveTCP=true) feature=Base
                  SuppressedNode
                    If barreno_actual≟3
                      barreno_actual := barreno_actual+1
                  internos := interpolate_pose(Linea17_A, Linea17_B, barreno_actual/barrenos_menos1)
                  Waypoint Waypoint (Variable): variable=internos
                  'desbaste_inicial'
                  bajada_broca := p[0,0,-0.024,0,0,0]
                  bajada := p[0,0,0.024,0,0,0]
                  MoveDirectionNode (selectedDirection=ZMinus toolParams=0.1, 0.15)
                    Until DISTANCE (allowActions=false deceleration=3 distanceNodeType=STOP) Distance=0.071; motionParameters(blendRadius=0)
                  MoveDirectionNode (selectedDirection=ZMinus toolParams=0.007, 0.007)
                    Until TOOL_CONTACT_DETECTION (allowActions=false retraction=0 decelerationAcceleration=0.02 decelerationAngularAcceleration=34.906585)
                  Popup Message (haltProgram=false message=punto contacto alanzdo inputType=Text)
                  MoveDirectionNode (selectedDirection=ZPlus toolParams=0.1, 0.15)
                    Until DISTANCE (allowActions=false deceleration=3 distanceNodeType=STOP) Distance=0.002; motionParameters(blendRadius=0)
                  Wait Sleep waitTime=0.3
                  Set DigitalOutput pin=config_out[1]; digitalValue=1
                  Wait Sleep waitTime=0.3
                  Loop Counting (count=1) loopVariable(name=Loop_137)
                    bajar := pose_add(get_actual_tcp_pose(), bajada_broca)
                    Waypoint Waypoint (Variable): motionParameters(jointSpeed=1.047198 jointAcceleration=1.396263 cartesianSpeed=0.004 cartesianAcceleration=0.004); variable=bajar
                    subir := pose_sub(get_actual_tcp_pose(), bajada_broca)
                    MoveDirectionNode (selectedDirection=ZPlus toolParams=0.015, 0.015)
                      Until DISTANCE (allowActions=false deceleration=3 distanceNodeType=STOP) Distance=0.002; motionParameters(blendRadius=0)
                    Set DigitalOutput pin=config_out[1]; digitalValue=0
                    Waypoint Waypoint (Variable): motionParameters(jointSpeed=1.047198 jointAcceleration=1.396263 cartesianSpeed=0.015 cartesianAcceleration=0.015); variable=subir
                    bajada_broca := pose_sub(bajada_broca, bajada)
                  MoveDirectionNode (selectedDirection=ZPlus toolParams=0.03, 0.035)
                    Until DISTANCE (allowActions=false deceleration=3 distanceNodeType=STOP) Distance=0.08; motionParameters(blendRadius=0)
                  Set DigitalOutput pin=config_out[1]; digitalValue=0
                  barreno_actual := barreno_actual+1
                  SuppressedNode
                    Call Quitar_broca
                  SuppressedNode
                    Call Poner_broca
        Popup Message (haltProgram=false message=Linea17 con chica Terminada! inputType=Text)
        Folder Linea18
          Folder Marcar_puntos
            MoveL speed 100 mm/s, acceleration 500 mm/s^2 (useActiveTCP=true) feature=Base
              Waypoint Linea18_A: TCP in base x=652.275 y=616.966 z=110.402 mm, rx=-1.5443 ry=-2.7321 rz=-0.0069 rad; joints [-149.578, -67.211, 98.412, -30.856, -279.791, 0.343] deg
              Folder bajada_comprobacion
                MoveDirectionNode (selectedDirection=ZMinus toolParams=0.1, 0.15)
                  Until DISTANCE (allowActions=false deceleration=3 distanceNodeType=STOP) Distance=0.071; motionParameters(blendRadius=0)
                MoveDirectionNode (selectedDirection=ZMinus toolParams=0.007, 0.007)
                  Until TOOL_CONTACT_DETECTION (allowActions=false retraction=0 decelerationAcceleration=0.02 decelerationAngularAcceleration=34.906585)
                MoveDirectionNode (selectedDirection=ZPlus toolParams=0.1, 0.15)
                  Until DISTANCE (allowActions=false deceleration=3 distanceNodeType=STOP) Distance=0.08; motionParameters(blendRadius=0)
              Waypoint Linea18_AB: TCP in base x=883.615 y=616.35 z=110.351 mm, rx=-1.5443 ry=-2.7321 rz=-0.0069 rad; joints [-156.916, -51.669, 73.431, -21.398, -287.108, 0.294] deg
              SuppressedNode
                Waypoint Linea18_B: TCP in base x=-1149.588 y=625.185 z=110.393 mm, rx=1.1641 ry=-2.9058 rz=0.0105 rad; joints [-36.247, -18.765, 11.523, 7.74, -268.979, 0.895] deg; TCP offset x=0.411 y=-218.298 z=37.994 mm, rx=1.558 ry=-0.1255 rz=0.1212 rad
              Folder bajada_comprobacion
                MoveDirectionNode (selectedDirection=ZMinus toolParams=0.1, 0.15)
                  Until DISTANCE (allowActions=false deceleration=3 distanceNodeType=STOP) Distance=0.071; motionParameters(blendRadius=0)
                MoveDirectionNode (selectedDirection=ZMinus toolParams=0.007, 0.007)
                  Until TOOL_CONTACT_DETECTION (allowActions=false retraction=0 decelerationAcceleration=0.02 decelerationAngularAcceleration=34.906585)
                MoveDirectionNode (selectedDirection=ZPlus toolParams=0.1, 0.15)
                  Until DISTANCE (allowActions=false deceleration=3 distanceNodeType=STOP) Distance=0.08; motionParameters(blendRadius=0)
          Folder AB
            'desbaste_inicial'
            bajada_broca := p[0,0,-0.008,0,0,0]
            barrenos_menos1 := 9
            barreno_actual := 0
            Loop While (checkContinuously=false) expression=barreno_actual≤barrenos_menos1
              Folder Perforacion
                MoveL speed 100 mm/s, acceleration 500 mm/s^2 (useActiveTCP=true) feature=Base
                  If barreno_actual≟6
                    barreno_actual := barreno_actual+1
                  internos := interpolate_pose(Linea18_A, Linea18_AB, barreno_actual/barrenos_menos1)
                  Waypoint Waypoint (Variable): variable=internos
                  'desbaste_inicial'
                  bajada_broca := p[0,0,-0.024,0,0,0]
                  bajada := p[0,0,0.024,0,0,0]
                  MoveDirectionNode (selectedDirection=ZMinus toolParams=0.1, 0.15)
                    Until DISTANCE (allowActions=false deceleration=3 distanceNodeType=STOP) Distance=0.071; motionParameters(blendRadius=0)
                  MoveDirectionNode (selectedDirection=ZMinus toolParams=0.007, 0.007)
                    Until TOOL_CONTACT_DETECTION (allowActions=false retraction=0 decelerationAcceleration=0.02 decelerationAngularAcceleration=34.906585)
                  Popup Message (haltProgram=false message=punto contacto alanzdo inputType=Text)
                  MoveDirectionNode (selectedDirection=ZPlus toolParams=0.015, 0.015)
                    Until DISTANCE (allowActions=false deceleration=3 distanceNodeType=STOP) Distance=0.007; motionParameters(blendRadius=0)
                  Wait Sleep waitTime=0.3
                  Set DigitalOutput pin=config_out[1]; digitalValue=1
                  Wait Sleep waitTime=0.3
                  Loop Counting (count=1) loopVariable(name=Loop_139)
                    bajar := pose_add(get_actual_tcp_pose(), bajada_broca)
                    Waypoint Waypoint (Variable): motionParameters(jointSpeed=1.047198 jointAcceleration=1.396263 cartesianSpeed=0.004 cartesianAcceleration=0.004); variable=bajar
                    subir := pose_sub(get_actual_tcp_pose(), bajada_broca)
                    MoveDirectionNode (selectedDirection=ZPlus toolParams=0.015, 0.015)
                      Until DISTANCE (allowActions=false deceleration=3 distanceNodeType=STOP) Distance=0.002; motionParameters(blendRadius=0)
                    Set DigitalOutput pin=config_out[1]; digitalValue=0
                    Waypoint Waypoint (Variable): motionParameters(jointSpeed=1.047198 jointAcceleration=1.396263 cartesianSpeed=0.015 cartesianAcceleration=0.015); variable=subir
                    bajada_broca := pose_sub(bajada_broca, bajada)
                  MoveDirectionNode (selectedDirection=ZPlus toolParams=0.1, 0.15)
                    Until DISTANCE (allowActions=false deceleration=3 distanceNodeType=STOP) Distance=0.08; motionParameters(blendRadius=0)
                  Set DigitalOutput pin=config_out[1]; digitalValue=0
                  barreno_actual := barreno_actual+1
                  Call Quitar_broca
                  Call Poner_broca
        Popup Message (haltProgram=false message=Linea18 con chica Terminada! inputType=Text)
        Folder Linea18B
          Folder Marcar_puntos
            MoveL speed 100 mm/s, acceleration 500 mm/s^2 (useActiveTCP=true) feature=Base
              Waypoint Linea18_BA: TCP in base x=909.905 y=616.222 z=110.421 mm, rx=-1.5443 ry=-2.7321 rz=-0.0069 rad; joints [-157.556, -49.622, 69.886, -19.898, -287.745, 0.289] deg; TCP offset x=0.411 y=-218.298 z=37.994 mm, rx=1.558 ry=-0.1255 rz=0.1212 rad
              Folder bajada_comprobacion
                MoveDirectionNode (selectedDirection=ZMinus toolParams=0.1, 0.15)
                  Until DISTANCE (allowActions=false deceleration=3 distanceNodeType=STOP) Distance=0.071; motionParameters(blendRadius=0)
                MoveDirectionNode (selectedDirection=ZMinus toolParams=0.007, 0.007)
                  Until TOOL_CONTACT_DETECTION (allowActions=false retraction=0 decelerationAcceleration=0.02 decelerationAngularAcceleration=34.906585)
                MoveDirectionNode (selectedDirection=ZPlus toolParams=0.1, 0.15)
                  Until DISTANCE (allowActions=false deceleration=3 distanceNodeType=STOP) Distance=0.08; motionParameters(blendRadius=0)
              SuppressedNode
                Waypoint Linea18_AB: TCP in base x=-890.203 y=626.114 z=110.875 mm, rx=-0.2145 ry=-3.1278 rz=-0.004 rad; joints [-38.182, -44.07, 60.007, -15.504, -219.471, 0.847] deg; TCP offset x=0.411 y=-218.298 z=37.994 mm, rx=1.558 ry=-0.1255 rz=0.1212 rad
              Waypoint Linea18_B referenceName=Linea18_B: TCP in base x=1141.235 y=615.792 z=110.308 mm, rx=-1.5443 ry=-2.7321 rz=-0.0069 rad; joints [-162.019, -22.381, 18.834, 3.929, -292.141, 0.256] deg; TCP offset x=0.411 y=-218.298 z=37.994 mm, rx=1.558 ry=-0.1255 rz=0.1212 rad
              Folder bajada_comprobacion
                MoveDirectionNode (selectedDirection=ZMinus toolParams=0.1, 0.15)
                  Until DISTANCE (allowActions=false deceleration=3 distanceNodeType=STOP) Distance=0.071; motionParameters(blendRadius=0)
                MoveDirectionNode (selectedDirection=ZMinus toolParams=0.007, 0.007)
                  Until TOOL_CONTACT_DETECTION (allowActions=false retraction=0 decelerationAcceleration=0.02 decelerationAngularAcceleration=34.906585)
                MoveDirectionNode (selectedDirection=ZPlus toolParams=0.1, 0.15)
                  Until DISTANCE (allowActions=false deceleration=3 distanceNodeType=STOP) Distance=0.08; motionParameters(blendRadius=0)
          Folder AB
            'desbaste_inicial'
            bajada_broca := p[0,0,-0.008,0,0,0]
            barrenos_menos1 := 9
            barreno_actual := 8
            Loop While (checkContinuously=false) expression=barreno_actual≤barrenos_menos1
              Folder Perforacion
                MoveL speed 100 mm/s, acceleration 500 mm/s^2 (useActiveTCP=true) feature=Base
                  If barreno_actual≟3
                    barreno_actual := barreno_actual+1
                  internos := interpolate_pose(Linea18_BA, Linea18_B, barreno_actual/barrenos_menos1)
                  Waypoint Waypoint (Variable): variable=internos
                  'desbaste_inicial'
                  bajada_broca := p[0,0,-0.024,0,0,0]
                  bajada := p[0,0,0.024,0,0,0]
                  MoveDirectionNode (selectedDirection=ZMinus toolParams=0.1, 0.15)
                    Until DISTANCE (allowActions=false deceleration=3 distanceNodeType=STOP) Distance=0.071; motionParameters(blendRadius=0)
                  MoveDirectionNode (selectedDirection=ZMinus toolParams=0.007, 0.007)
                    Until TOOL_CONTACT_DETECTION (allowActions=false retraction=0 decelerationAcceleration=0.02 decelerationAngularAcceleration=34.906585)
                  Popup Message (haltProgram=false message=punto contacto alanzdo inputType=Text)
                  MoveDirectionNode (selectedDirection=ZPlus toolParams=0.015, 0.015)
                    Until DISTANCE (allowActions=false deceleration=3 distanceNodeType=STOP) Distance=0.007; motionParameters(blendRadius=0)
                  Wait Sleep waitTime=0.3
                  Set DigitalOutput pin=config_out[1]; digitalValue=1
                  Wait Sleep waitTime=0.3
                  Loop Counting (count=1) loopVariable(name=Loop_28)
                    bajar := pose_add(get_actual_tcp_pose(), bajada_broca)
                    Waypoint Waypoint (Variable): motionParameters(jointSpeed=1.047198 jointAcceleration=1.396263 cartesianSpeed=0.004 cartesianAcceleration=0.004); variable=bajar
                    subir := pose_sub(get_actual_tcp_pose(), bajada_broca)
                    MoveDirectionNode (selectedDirection=ZPlus toolParams=0.015, 0.015)
                      Until DISTANCE (allowActions=false deceleration=3 distanceNodeType=STOP) Distance=0.002; motionParameters(blendRadius=0)
                    Set DigitalOutput pin=config_out[1]; digitalValue=0
                    Waypoint Waypoint (Variable): motionParameters(jointSpeed=1.047198 jointAcceleration=1.396263 cartesianSpeed=0.015 cartesianAcceleration=0.015); variable=subir
                    bajada_broca := pose_sub(bajada_broca, bajada)
                  MoveDirectionNode (selectedDirection=ZPlus toolParams=0.1, 0.15)
                    Until DISTANCE (allowActions=false deceleration=3 distanceNodeType=STOP) Distance=0.08; motionParameters(blendRadius=0)
                  Set DigitalOutput pin=config_out[1]; digitalValue=0
                  barreno_actual := barreno_actual+1
                  Call Quitar_broca
                  Call Poner_broca
        Popup Message (haltProgram=false message=Linea18B con chica Terminada! inputType=Text)
      cambiar_broca := True
      SuppressedNode
        Call Quitar_broca
      SuppressedNode
        Call Poner_broca
      SuppressedNode
        Folder Broca_2
          Folder Linea7
            Folder Marcar_puntos
              MoveL speed 100 mm/s, acceleration 500 mm/s^2 (useActiveTCP=true) feature=Base
                Waypoint Home2: TCP in base x=-476.229 y=0 z=568.737 mm, rx=2.0263 ry=-2.3929 rz=-0.0208 rad; joints [-32.551, -116.469, 98.413, 17.843, -302.102, -0.163] deg; TCP offset x=0.411 y=-218.298 z=37.994 mm, rx=1.558 ry=-0.1255 rz=0.1212 rad
                Waypoint Linea7_A: TCP in base x=-749.561 y=-351.839 z=110.843 mm, rx=3.1084 ry=-0.3759 rz=-0.0174 rad; joints [1.917, -65.95, 96.598, -30.808, -353.455, -0.309] deg
                Folder bajada_comprobacion
                  MoveDirectionNode (selectedDirection=ZMinus toolParams=0.1, 0.15)
                    Until DISTANCE (allowActions=false deceleration=3 distanceNodeType=STOP) Distance=0.071; motionParameters(blendRadius=0)
                  MoveDirectionNode (selectedDirection=ZMinus toolParams=0.007, 0.007)
                    Until TOOL_CONTACT_DETECTION (allowActions=false retraction=0 decelerationAcceleration=0.007 decelerationAngularAcceleration=34.906585)
                  MoveDirectionNode (selectedDirection=ZPlus toolParams=0.1, 0.15)
                    Until DISTANCE (allowActions=false deceleration=3 distanceNodeType=STOP) Distance=0.08; motionParameters(blendRadius=0)
                Waypoint Linea7_B: TCP in base x=-795.37 y=-351.638 z=110.748 mm, rx=3.1084 ry=-0.3758 rz=-0.0174 rad; joints [1.792, -62.243, 90.906, -28.822, -353.578, -0.309] deg
                Folder bajada_comprobacion
                  MoveDirectionNode (selectedDirection=ZMinus toolParams=0.1, 0.15)
                    Until DISTANCE (allowActions=false deceleration=3 distanceNodeType=STOP) Distance=0.071; motionParameters(blendRadius=0)
                  MoveDirectionNode (selectedDirection=ZMinus toolParams=0.007, 0.007)
                    Until TOOL_CONTACT_DETECTION (allowActions=false retraction=0 decelerationAcceleration=0.007 decelerationAngularAcceleration=34.906585)
                  MoveDirectionNode (selectedDirection=ZPlus toolParams=0.1, 0.15)
                    Until DISTANCE (allowActions=false deceleration=3 distanceNodeType=STOP) Distance=0.08; motionParameters(blendRadius=0)
            Folder AB
              'desbaste_inicial'
              bajada_broca := p[0,0,-0.008,0,0,0]
              barrenos_menos1 := 2
              barreno_actual := 0
              Loop While (checkContinuously=false) expression=barreno_actual≤barrenos_menos1
                Folder Perforacion
                  MoveL speed 100 mm/s, acceleration 500 mm/s^2 (useActiveTCP=true) feature=Base
                    internos := interpolate_pose(Linea7_A, Linea7_B, barreno_actual/barrenos_menos1)
                    Waypoint Waypoint (Variable): variable=internos
                    'desbaste_inicial'
                    bajada_broca := p[0,0,-0.024,0,0,0]
                    bajada := p[0,0,0.024,0,0,0]
                    MoveDirectionNode (selectedDirection=ZMinus toolParams=0.1, 0.15)
                      Until DISTANCE (allowActions=false deceleration=3 distanceNodeType=STOP) Distance=0.071; motionParameters(blendRadius=0)
                    MoveDirectionNode (selectedDirection=ZMinus toolParams=0.01, 0.01)
                      Until TOOL_CONTACT_DETECTION (allowActions=false retraction=0 decelerationAcceleration=0.01 decelerationAngularAcceleration=34.906585)
                    Popup Message (haltProgram=false message=punto contacto alanzdo inputType=Text)
                    MoveDirectionNode (selectedDirection=ZPlus toolParams=0.003, 0.005)
                      Until DISTANCE (allowActions=false deceleration=3 distanceNodeType=STOP) Distance=0.002; motionParameters(blendRadius=0)
                    Wait Sleep waitTime=0.3
                    Set DigitalOutput pin=config_out[1]; digitalValue=1
                    Wait Sleep waitTime=0.3
                    Loop Counting (count=1) loopVariable(name=Loop_47)
                      bajar := pose_add(get_actual_tcp_pose(), bajada_broca)
                      Waypoint Waypoint (Variable): motionParameters(jointSpeed=1.047198 jointAcceleration=1.396263 cartesianSpeed=0.001 cartesianAcceleration=0.005); variable=bajar
                      subir := pose_sub(get_actual_tcp_pose(), bajada_broca)
                      Waypoint Waypoint (Variable): motionParameters(jointSpeed=1.047198 jointAcceleration=1.396263 cartesianSpeed=0.005 cartesianAcceleration=0.01); variable=subir
                      bajada_broca := pose_sub(bajada_broca, bajada)
                    MoveDirectionNode (selectedDirection=ZPlus toolParams=0.1, 0.15)
                      Until DISTANCE (allowActions=false deceleration=3 distanceNodeType=STOP) Distance=0.08; motionParameters(blendRadius=0)
                    Set DigitalOutput pin=config_out[1]; digitalValue=0
                    barreno_actual := barreno_actual+1
                    Call Quitar_broca
                    Call Poner_broca
          Popup Message (haltProgram=false message=Linea7 con chica Terminada! inputType=Text)
          Folder Linea8
            Folder Marcar_puntos
              MoveL speed 100 mm/s, acceleration 500 mm/s^2 (useActiveTCP=true) feature=Base
                Waypoint Linea8_A: TCP in base x=-897.665 y=-351.421 z=110.406 mm, rx=3.1084 ry=-0.3758 rz=-0.0174 rad; joints [1.574, -53.621, 76.868, -23.4, -353.783, -0.317] deg; TCP offset x=0.411 y=-218.298 z=37.994 mm, rx=1.558 ry=-0.1255 rz=0.1212 rad
                Folder bajada_comprobacion
                  MoveDirectionNode (selectedDirection=ZMinus toolParams=0.1, 0.15)
                    Until DISTANCE (allowActions=false deceleration=3 distanceNodeType=STOP) Distance=0.071; motionParameters(blendRadius=0)
                  MoveDirectionNode (selectedDirection=ZMinus toolParams=0.007, 0.007)
                    Until TOOL_CONTACT_DETECTION (allowActions=false retraction=0 decelerationAcceleration=0.007 decelerationAngularAcceleration=34.906585)
                  MoveDirectionNode (selectedDirection=ZPlus toolParams=0.1, 0.15)
                    Until DISTANCE (allowActions=false deceleration=3 distanceNodeType=STOP) Distance=0.08; motionParameters(blendRadius=0)
                Waypoint Linea8_B: TCP in base x=-1021.743 y=-350.913 z=110.77 mm, rx=3.1084 ry=-0.3758 rz=-0.0173 rad; joints [1.351, -41.656, 55.75, -14.225, -353.984, -0.335] deg; TCP offset x=0.411 y=-218.298 z=37.994 mm, rx=1.558 ry=-0.1255 rz=0.1212 rad
                Folder bajada_comprobacion
                  MoveDirectionNode (selectedDirection=ZMinus toolParams=0.1, 0.15)
                    Until DISTANCE (allowActions=false deceleration=3 distanceNodeType=STOP) Distance=0.071; motionParameters(blendRadius=0)
                  MoveDirectionNode (selectedDirection=ZMinus toolParams=0.007, 0.007)
                    Until TOOL_CONTACT_DETECTION (allowActions=false retraction=0 decelerationAcceleration=0.007 decelerationAngularAcceleration=34.906585)
                  MoveDirectionNode (selectedDirection=ZPlus toolParams=0.1, 0.15)
                    Until DISTANCE (allowActions=false deceleration=3 distanceNodeType=STOP) Distance=0.08; motionParameters(blendRadius=0)
            Folder AB
              'desbaste_inicial'
              bajada_broca := p[0,0,-0.008,0,0,0]
              barrenos_menos1 := 5
              barreno_actual := 0
              Loop While (checkContinuously=false) expression=barreno_actual≤barrenos_menos1
                Folder Perforacion
                  MoveL speed 100 mm/s, acceleration 500 mm/s^2 (useActiveTCP=true) feature=Base
                    internos := interpolate_pose(Linea8_A, Linea8_B, barreno_actual/barrenos_menos1)
                    Waypoint Waypoint (Variable): variable=internos
                    'desbaste_inicial'
                    bajada_broca := p[0,0,-0.024,0,0,0]
                    bajada := p[0,0,0.0024,0,0,0]
                    MoveDirectionNode (selectedDirection=ZMinus toolParams=0.1, 0.15)
                      Until DISTANCE (allowActions=false deceleration=3 distanceNodeType=STOP) Distance=0.071; motionParameters(blendRadius=0)
                    MoveDirectionNode (selectedDirection=ZMinus toolParams=0.01, 0.01)
                      Until TOOL_CONTACT_DETECTION (allowActions=false retraction=0 decelerationAcceleration=0.01 decelerationAngularAcceleration=34.906585)
                    Popup Message (haltProgram=false message=punto contacto alanzdo inputType=Text)
                    MoveDirectionNode (selectedDirection=ZPlus toolParams=0.003, 0.005)
                      Until DISTANCE (allowActions=false deceleration=3 distanceNodeType=STOP) Distance=0.002; motionParameters(blendRadius=0)
                    Wait Sleep waitTime=0.3
                    Set DigitalOutput pin=config_out[1]; digitalValue=1
                    Wait Sleep waitTime=0.3
                    Loop Counting (count=1) loopVariable(name=Loop_53)
                      bajar := pose_add(get_actual_tcp_pose(), bajada_broca)
                      Waypoint Waypoint (Variable): motionParameters(jointSpeed=1.047198 jointAcceleration=1.396263 cartesianSpeed=0.001 cartesianAcceleration=0.005); variable=bajar
                      subir := pose_sub(get_actual_tcp_pose(), bajada_broca)
                      Waypoint Waypoint (Variable): motionParameters(jointSpeed=1.047198 jointAcceleration=1.396263 cartesianSpeed=0.005 cartesianAcceleration=0.01); variable=subir
                      bajada_broca := pose_sub(bajada_broca, bajada)
                    MoveDirectionNode (selectedDirection=ZPlus toolParams=0.1, 0.15)
                      Until DISTANCE (allowActions=false deceleration=3 distanceNodeType=STOP) Distance=0.08; motionParameters(blendRadius=0)
                    Set DigitalOutput pin=config_out[1]; digitalValue=0
                    barreno_actual := barreno_actual+1
                    Call Quitar_broca
                    Call Poner_broca
          Popup Message (haltProgram=false message=Linea8 con chica Terminada! inputType=Text)
          Folder Linea9
            Folder Marcar_puntos
              MoveL speed 100 mm/s, acceleration 500 mm/s^2 (useActiveTCP=true) feature=Base
                Waypoint Linea9_A: TCP in base x=-1101.64 y=-350.63 z=110.828 mm, rx=3.1084 ry=-0.3759 rz=-0.0174 rad; joints [1.234, -31.471, 36.669, -5.317, -354.073, -0.351] deg; TCP offset x=0.411 y=-218.298 z=37.994 mm, rx=1.558 ry=-0.1255 rz=0.1212 rad
                Folder bajada_comprobacion
                  MoveDirectionNode (selectedDirection=ZMinus toolParams=0.1, 0.15)
                    Until DISTANCE (allowActions=false deceleration=3 distanceNodeType=STOP) Distance=0.071; motionParameters(blendRadius=0)
                  MoveDirectionNode (selectedDirection=ZMinus toolParams=0.007, 0.007)
                    Until TOOL_CONTACT_DETECTION (allowActions=false retraction=0 decelerationAcceleration=0.007 decelerationAngularAcceleration=34.906585)
                  MoveDirectionNode (selectedDirection=ZPlus toolParams=0.1, 0.15)
                    Until DISTANCE (allowActions=false deceleration=3 distanceNodeType=STOP) Distance=0.08; motionParameters(blendRadius=0)
                Waypoint Linea9_B: TCP in base x=-1151.202 y=-350.816 z=110.405 mm, rx=3.1084 ry=-0.3759 rz=-0.0174 rad; joints [1.184, -21.077, 16.327, 4.623, -354.093, -0.341] deg
                Folder bajada_comprobacion
                  MoveDirectionNode (selectedDirection=ZMinus toolParams=0.1, 0.15)
                    Until DISTANCE (allowActions=false deceleration=3 distanceNodeType=STOP) Distance=0.071; motionParameters(blendRadius=0)
                  MoveDirectionNode (selectedDirection=ZMinus toolParams=0.007, 0.007)
                    Until TOOL_CONTACT_DETECTION (allowActions=false retraction=0 decelerationAcceleration=0.007 decelerationAngularAcceleration=34.906585)
                  MoveDirectionNode (selectedDirection=ZPlus toolParams=0.1, 0.15)
                    Until DISTANCE (allowActions=false deceleration=3 distanceNodeType=STOP) Distance=0.08; motionParameters(blendRadius=0)
            Folder AB
              'desbaste_inicial'
              bajada_broca := p[0,0,-0.008,0,0,0]
              barrenos_menos1 := 2
              barreno_actual := 0
              Loop While (checkContinuously=false) expression=barreno_actual≤barrenos_menos1
                Folder Perforacion
                  MoveL speed 100 mm/s, acceleration 500 mm/s^2 (useActiveTCP=true) feature=Base
                    internos := interpolate_pose(Linea9_A, Linea9_B, barreno_actual/barrenos_menos1)
                    Waypoint Waypoint (Variable): variable=internos
                    'desbaste_inicial'
                    bajada_broca := p[0,0,-0.024,0,0,0]
                    bajada := p[0,0,0.024,0,0,0]
                    MoveDirectionNode (selectedDirection=ZMinus toolParams=0.1, 0.15)
                      Until DISTANCE (allowActions=false deceleration=3 distanceNodeType=STOP) Distance=0.071; motionParameters(blendRadius=0)
                    MoveDirectionNode (selectedDirection=ZMinus toolParams=0.01, 0.01)
                      Until TOOL_CONTACT_DETECTION (allowActions=false retraction=0 decelerationAcceleration=0.01 decelerationAngularAcceleration=34.906585)
                    Popup Message (haltProgram=false message=punto contacto alanzdo inputType=Text)
                    MoveDirectionNode (selectedDirection=ZPlus toolParams=0.003, 0.005)
                      Until DISTANCE (allowActions=false deceleration=3 distanceNodeType=STOP) Distance=0.002; motionParameters(blendRadius=0)
                    Wait Sleep waitTime=0.3
                    Set DigitalOutput pin=config_out[1]; digitalValue=1
                    Wait Sleep waitTime=0.3
                    Loop Counting (count=1) loopVariable=Loop_56
                      bajar := pose_add(get_actual_tcp_pose(), bajada_broca)
                      Waypoint Waypoint (Variable): motionParameters(jointSpeed=1.047198 jointAcceleration=1.396263 cartesianSpeed=0.001 cartesianAcceleration=0.005); variable=bajar
                      subir := pose_sub(get_actual_tcp_pose(), bajada_broca)
                      Waypoint Waypoint (Variable): motionParameters(jointSpeed=1.047198 jointAcceleration=1.396263 cartesianSpeed=0.005 cartesianAcceleration=0.01); variable=subir
                      bajada_broca := pose_sub(bajada_broca, bajada)
                    MoveDirectionNode (selectedDirection=ZPlus toolParams=0.1, 0.15)
                      Until DISTANCE (allowActions=false deceleration=3 distanceNodeType=STOP) Distance=0.08; motionParameters(blendRadius=0)
                    Set DigitalOutput pin=config_out[1]; digitalValue=0
                    barreno_actual := barreno_actual+1
                    Call Quitar_broca
                    Call Poner_broca
          Popup Message (haltProgram=false message=Linea9 con chica Terminada! inputType=Text)
          Folder Linea10
            Folder Marcar_puntos
              MoveL speed 100 mm/s, acceleration 500 mm/s^2 (useActiveTCP=true) feature=Base
                Waypoint Home2: TCP in base x=-476.229 y=0 z=568.737 mm, rx=2.0263 ry=-2.3929 rz=-0.0208 rad; joints [-32.551, -116.469, 98.413, 17.843, -302.102, -0.163] deg; TCP offset x=0.411 y=-218.298 z=37.994 mm, rx=1.558 ry=-0.1255 rz=0.1212 rad
                Waypoint Linea10_A: TCP in base x=-633.044 y=-316.972 z=110.617 mm, rx=3.1084 ry=-0.3759 rz=-0.0173 rad; joints [-0.95, -76.145, 111.037, -35.154, -356.326, -0.202] deg; TCP offset x=0.411 y=-218.298 z=37.994 mm, rx=1.558 ry=-0.1255 rz=0.1212 rad
                Folder bajada_comprobacion
                  MoveDirectionNode (selectedDirection=ZMinus toolParams=0.1, 0.15)
                    Until DISTANCE (allowActions=false deceleration=3 distanceNodeType=STOP) Distance=0.071; motionParameters(blendRadius=0)
                  MoveDirectionNode (selectedDirection=ZMinus toolParams=0.007, 0.007)
                    Until TOOL_CONTACT_DETECTION (allowActions=false retraction=0 decelerationAcceleration=0.007 decelerationAngularAcceleration=34.906585)
                  MoveDirectionNode (selectedDirection=ZPlus toolParams=0.1, 0.15)
                    Until DISTANCE (allowActions=false deceleration=3 distanceNodeType=STOP) Distance=0.08; motionParameters(blendRadius=0)
                Waypoint Linea10_B: TCP in base x=-636.724 y=-267.195 z=110.576 mm, rx=2.0205 ry=-2.3939 rz=-0.0206 rad; joints [10.728, -83.916, 120.692, -37.175, -258.773, -0.177] deg
                Folder bajada_comprobacion
                  MoveDirectionNode (selectedDirection=ZMinus toolParams=0.1, 0.15)
                    Until DISTANCE (allowActions=false deceleration=3 distanceNodeType=STOP) Distance=0.071; motionParameters(blendRadius=0)
                  MoveDirectionNode (selectedDirection=ZMinus toolParams=0.007, 0.007)
                    Until TOOL_CONTACT_DETECTION (allowActions=false retraction=0 decelerationAcceleration=0.007 decelerationAngularAcceleration=34.906585)
                  MoveDirectionNode (selectedDirection=ZPlus toolParams=0.1, 0.15)
                    Until DISTANCE (allowActions=false deceleration=3 distanceNodeType=STOP) Distance=0.08; motionParameters(blendRadius=0)
            Folder AB
              'desbaste_inicial'
              bajada_broca := p[0,0,-0.008,0,0,0]
              barrenos_menos1 := 2
              barreno_actual := 0
              Loop While (checkContinuously=false) expression=barreno_actual≤barrenos_menos1
                Folder Perforacion
                  MoveL speed 100 mm/s, acceleration 500 mm/s^2 (useActiveTCP=true) feature=Base
                    internos := interpolate_pose(Linea10_A, Linea10_B, barreno_actual/barrenos_menos1)
                    Waypoint Waypoint (Variable): variable=internos
                    'desbaste_inicial'
                    bajada_broca := p[0,0,-0.024,0,0,0]
                    bajada := p[0,0,0.024,0,0,0]
                    MoveDirectionNode (selectedDirection=ZMinus toolParams=0.1, 0.15)
                      Until DISTANCE (allowActions=false deceleration=3 distanceNodeType=STOP) Distance=0.071; motionParameters(blendRadius=0)
                    MoveDirectionNode (selectedDirection=ZMinus toolParams=0.001, 0.001)
                      Until TOOL_CONTACT_DETECTION (allowActions=false retraction=0 decelerationAcceleration=0.001 decelerationAngularAcceleration=34.906585)
                    Popup Message (haltProgram=false message=punto contacto alanzdo inputType=Text)
                    MoveDirectionNode (selectedDirection=ZPlus toolParams=0.003, 0.005)
                      Until DISTANCE (allowActions=false deceleration=3 distanceNodeType=STOP) Distance=0.002; motionParameters(blendRadius=0)
                    Wait Sleep waitTime=0.3
                    Set DigitalOutput pin=config_out[1]; digitalValue=1
                    Wait Sleep waitTime=0.3
                    Loop Counting (count=1) loopVariable(name=Loop_58)
                      bajar := pose_add(get_actual_tcp_pose(), bajada_broca)
                      Waypoint Waypoint (Variable): motionParameters(jointSpeed=1.047198 jointAcceleration=1.396263 cartesianSpeed=0.001 cartesianAcceleration=0.005); variable=bajar
                      subir := pose_sub(get_actual_tcp_pose(), bajada_broca)
                      Waypoint Waypoint (Variable): motionParameters(jointSpeed=1.047198 jointAcceleration=1.396263 cartesianSpeed=0.005 cartesianAcceleration=0.01); variable=subir
                      bajada_broca := pose_sub(bajada_broca, bajada)
                    MoveDirectionNode (selectedDirection=ZPlus toolParams=0.1, 0.15)
                      Until DISTANCE (allowActions=false deceleration=3 distanceNodeType=STOP) Distance=0.08; motionParameters(blendRadius=0)
                    Set DigitalOutput pin=config_out[1]; digitalValue=0
                    barreno_actual := barreno_actual+1
                    Call Quitar_broca
                    Call Poner_broca
          Popup Message (haltProgram=false message=Linea10 con chica Terminada! inputType=Text)
          Folder Linea11
            Folder Marcar_puntos
              MoveL speed 100 mm/s, acceleration 500 mm/s^2 (useActiveTCP=true) feature=Base
                Waypoint Linea11_A: TCP in base x=-636.133 y=-137.915 z=110.44 mm, rx=2.0204 ry=-2.394 rz=-0.0205 rad; joints [-4.201, -88.707, 125.915, -37.584, -273.698, -0.078] deg
                Folder bajada_comprobacion
                  MoveDirectionNode (selectedDirection=ZMinus toolParams=0.1, 0.15)
                    Until DISTANCE (allowActions=false deceleration=3 distanceNodeType=STOP) Distance=0.071; motionParameters(blendRadius=0)
                  MoveDirectionNode (selectedDirection=ZMinus toolParams=0.007, 0.007)
                    Until TOOL_CONTACT_DETECTION (allowActions=false retraction=0 decelerationAcceleration=0.007 decelerationAngularAcceleration=34.906585)
                  MoveDirectionNode (selectedDirection=ZPlus toolParams=0.1, 0.15)
                    Until DISTANCE (allowActions=false deceleration=3 distanceNodeType=STOP) Distance=0.08; motionParameters(blendRadius=0)
                Waypoint Linea11_B: TCP in base x=-635.407 y=-82.609 z=110.403 mm, rx=2.0204 ry=-2.3939 rz=-0.0206 rad; joints [-11.006, -90.015, 127.249, -37.609, -280.504, -0.032] deg
                Folder bajada_comprobacion
                  MoveDirectionNode (selectedDirection=ZMinus toolParams=0.1, 0.15)
                    Until DISTANCE (allowActions=false deceleration=3 distanceNodeType=STOP) Distance=0.071; motionParameters(blendRadius=0)
                  MoveDirectionNode (selectedDirection=ZMinus toolParams=0.007, 0.007)
                    Until TOOL_CONTACT_DETECTION (allowActions=false retraction=0 decelerationAcceleration=0.007 decelerationAngularAcceleration=34.906585)
                  MoveDirectionNode (selectedDirection=ZPlus toolParams=0.1, 0.15)
                    Until DISTANCE (allowActions=false deceleration=3 distanceNodeType=STOP) Distance=0.08; motionParameters(blendRadius=0)
            Folder AB
              'desbaste_inicial'
              bajada_broca := p[0,0,-0.008,0,0,0]
              barrenos_menos1 := 2
              barreno_actual := 0
              Loop While (checkContinuously=false) expression=barreno_actual≤barrenos_menos1
                Folder Perforacion
                  MoveL speed 100 mm/s, acceleration 500 mm/s^2 (useActiveTCP=true) feature=Base
                    SuppressedNode
                      If barreno_actual≟5
                        barreno_actual := barreno_actual+1
                    internos := interpolate_pose(Linea11_A, Linea11_B, barreno_actual/barrenos_menos1)
                    Waypoint Waypoint (Variable): variable=internos
                    'desbaste_inicial'
                    bajada_broca := p[0,0,-0.024,0,0,0]
                    bajada := p[0,0,0.024,0,0,0]
                    MoveDirectionNode (selectedDirection=ZMinus toolParams=0.1, 0.15)
                      Until DISTANCE (allowActions=false deceleration=3 distanceNodeType=STOP) Distance=0.071; motionParameters(blendRadius=0)
                    MoveDirectionNode (selectedDirection=ZMinus toolParams=0.001, 0.001)
                      Until TOOL_CONTACT_DETECTION (allowActions=false retraction=0 decelerationAcceleration=0.001 decelerationAngularAcceleration=34.906585)
                    Popup Message (haltProgram=false message=punto contacto alanzdo inputType=Text)
                    MoveDirectionNode (selectedDirection=ZPlus toolParams=0.003, 0.005)
                      Until DISTANCE (allowActions=false deceleration=3 distanceNodeType=STOP) Distance=0.002; motionParameters(blendRadius=0)
                    Wait Sleep waitTime=0.3
                    Set DigitalOutput pin=config_out[1]; digitalValue=1
                    Wait Sleep waitTime=0.3
                    Loop Counting (count=1) loopVariable=Loop_74
                      bajar := pose_add(get_actual_tcp_pose(), bajada_broca)
                      Waypoint Waypoint (Variable): motionParameters(jointSpeed=1.047198 jointAcceleration=1.396263 cartesianSpeed=0.001 cartesianAcceleration=0.005); variable=bajar
                      subir := pose_sub(get_actual_tcp_pose(), bajada_broca)
                      Waypoint Waypoint (Variable): motionParameters(jointSpeed=1.047198 jointAcceleration=1.396263 cartesianSpeed=0.005 cartesianAcceleration=0.01); variable=subir
                      bajada_broca := pose_sub(bajada_broca, bajada)
                    MoveDirectionNode (selectedDirection=ZPlus toolParams=0.1, 0.15)
                      Until DISTANCE (allowActions=false deceleration=3 distanceNodeType=STOP) Distance=0.08; motionParameters(blendRadius=0)
                    Set DigitalOutput pin=config_out[1]; digitalValue=0
                    barreno_actual := barreno_actual+1
                    Call Quitar_broca
                    Call Poner_broca
          Popup Message (haltProgram=false message=Linea11 con chica Terminada! inputType=Text)
          Folder Linea12
            Folder Marcar_puntos
              MoveL speed 100 mm/s, acceleration 500 mm/s^2 (useActiveTCP=true) feature=Base
                Waypoint Linea12_A: TCP in base x=-635.979 y=-59.028 z=110.553 mm, rx=2.0204 ry=-2.3939 rz=-0.0205 rad; joints [-13.896, -90.321, 127.534, -37.586, -283.394, -0.016] deg
                Folder bajada_comprobacion
                  MoveDirectionNode (selectedDirection=ZMinus toolParams=0.1, 0.15)
                    Until DISTANCE (allowActions=false deceleration=3 distanceNodeType=STOP) Distance=0.071; motionParameters(blendRadius=0)
                  MoveDirectionNode (selectedDirection=ZMinus toolParams=0.007, 0.007)
                    Until TOOL_CONTACT_DETECTION (allowActions=false retraction=0 decelerationAcceleration=0.007 decelerationAngularAcceleration=34.906585)
                  MoveDirectionNode (selectedDirection=ZPlus toolParams=0.1, 0.15)
                    Until DISTANCE (allowActions=false deceleration=3 distanceNodeType=STOP) Distance=0.08; motionParameters(blendRadius=0)
                Waypoint Linea12_B: TCP in base x=-634.713 y=114.271 z=110.459 mm, rx=2.0204 ry=-2.3939 rz=-0.0206 rad; joints [-33.928, -89.524, 126.748, -37.639, -303.428, 0.135] deg
                Folder bajada_comprobacion
                  MoveDirectionNode (selectedDirection=ZMinus toolParams=0.1, 0.15)
                    Until DISTANCE (allowActions=false deceleration=3 distanceNodeType=STOP) Distance=0.071; motionParameters(blendRadius=0)
                  MoveDirectionNode (selectedDirection=ZMinus toolParams=0.007, 0.007)
                    Until TOOL_CONTACT_DETECTION (allowActions=false retraction=0 decelerationAcceleration=0.007 decelerationAngularAcceleration=34.906585)
                  MoveDirectionNode (selectedDirection=ZPlus toolParams=0.1, 0.15)
                    Until DISTANCE (allowActions=false deceleration=3 distanceNodeType=STOP) Distance=0.08; motionParameters(blendRadius=0)
            Folder AB
              'desbaste_inicial'
              bajada_broca := p[0,0,-0.008,0,0,0]
              barrenos_menos1 := 7
              barreno_actual := 0
              Loop While (checkContinuously=false) expression=barreno_actual≤barrenos_menos1
                Folder Perforacion
                  MoveL speed 100 mm/s, acceleration 500 mm/s^2 (useActiveTCP=true) feature=Base
                    If barreno_actual≟2
                      barreno_actual := barreno_actual+1
                    internos := interpolate_pose(Linea12_A, Linea12_B, barreno_actual/barrenos_menos1)
                    Waypoint Waypoint (Variable): variable=internos
                    'desbaste_inicial'
                    bajada_broca := p[0,0,-0.024,0,0,0]
                    bajada := p[0,0,0.024,0,0,0]
